LIN {X 0,Y 383.396,Z 1180.828,A -85,B 0,C 180,E1 16065.026,E2 16065.026} C_VEL
LIN {X 0,Y 390.535,Z 1171.867,A -85,B 0,C 180,E1 16063.935,E2 16063.935} C_VEL
LIN {X 0,Y 376.385,Z 1188.469,A -85,B 0,C 180,E1 16061.413,E2 16061.413} C_VEL
LIN {X 0,Y 362.666,Z 1204.614,A -85,B 0,C 180,E1 16058.341,E2 16058.341} C_VEL
LIN {X 0,Y 350.721,Z 1218.775,A -85,B 0,C 180,E1 16054.963,E2 16054.963} C_VEL
LIN {X 0,Y 340.496,Z 1230.965,A -85,B 0,C 180,E1 16051.317,E2 16051.317} C_VEL
LIN {X 0,Y 331.986,Z 1241.186,A -85,B 0,C 180,E1 16047.44,E2 16047.44} C_VEL
LIN {X 0,Y 325.156,Z 1249.467,A -85,B 0,C 180,E1 16043.371,E2 16043.371} C_VEL
LIN {X 0,Y 320.144,Z 1255.613,A -85,B 0,C 180,E1 16039.333,E2 16039.333} C_VEL
LIN {X 0,Y 316.54,Z 1259.979,A -85,B 0,C 180,E1 16035.2,E2 16035.2} C_VEL
LIN {X 0,Y 314.272,Z 1262.44,A -85,B 0,C 180,E1 16031.191,E2 16031.191} C_VEL
LIN {X 0,Y 312.948,Z 1263.309,A -85,B 0,C 180,E1 16026.974,E2 16026.974} C_VEL
LIN {X 0,Y 312.379,Z 1262.543,A -85,B 0,C 180,E1 16023.119,E2 16023.119} C_VEL
LIN {X 0,Y 312.208,Z 1260.385,A -85,B 0,C 180,E1 16019.633,E2 16019.633} C_VEL
LIN {X 0,Y 312.174,Z 1256.694,A -85,B 0,C 180,E1 16015.959,E2 16015.959} C_VEL
LIN {X 0,Y 312.386,Z 1251.681,A -85,B 0,C 180,E1 16012.459,E2 16012.459} C_VEL
LIN {X 0,Y 312.913,Z 1245.037,A -85,B 0,C 180,E1 16008.946,E2 16008.946} C_VEL
LIN {X 0,Y 313.943,Z 1236.737,A -85,B 0,C 180,E1 16005.427,E2 16005.427} C_VEL
LIN {X 0,Y 315.598,Z 1226.498,A -85,B 0,C 180,E1 16001.897,E2 16001.897} C_VEL
LIN {X 0,Y 317.811,Z 1214.873,A -85,B 0,C 180,E1 15998.595,E2 15998.595} C_VEL
LIN {X 0,Y 320.732,Z 1201.077,A -85,B 0,C 180,E1 15995.307,E2 15995.307} C_VEL
LIN {X 0,Y 324.178,Z 1185.749,A -85,B 0,C 180,E1 15992.242,E2 15992.242} C_VEL
LIN {X 0,Y 327.919,Z 1169.466,A -85,B 0,C 180,E1 15989.49,E2 15989.49} C_VEL
LIN {X 0,Y 332.099,Z 1150.975,A -85,B 0,C 180,E1 15986.862,E2 15986.862} C_VEL
LIN {X 0,Y 336.467,Z 1130.85,A -85,B 0,C 180,E1 15984.481,E2 15984.481} C_VEL
LIN {X 0,Y 340.596,Z 1110.333,A -85,B 0,C 180,E1 15982.46,E2 15982.46} C_VEL
LIN {X 0,Y 344.502,Z 1089.321,A -85,B 0,C 180,E1 15980.748,E2 15980.748} C_VEL
LIN {X 0,Y 348.276,Z 1066.302,A -85,B 0,C 180,E1 15979.221,E2 15979.221} C_VEL
LIN {X 0,Y 351.6,Z 1042.308,A -85,B 0,C 180,E1 15977.965,E2 15977.965} C_VEL
LIN {X 0,Y 354.32,Z 1018.528,A -85,B 0,C 180,E1 15977.027,E2 15977.027} C_VEL
LIN {X 0,Y 373.54,Z 802.907,A -85,B 0,C 180,E1 15971.161,E2 15971.161} C_VEL
LIN {X 0,Y 358.853,Z 773.867,A -85,B 0,C 180,E1 15968.29,E2 15968.29} C_VEL
LIN {X 0,Y 344.851,Z 748.162,A -85,B 0,C 180,E1 15965.343,E2 15965.343} C_VEL
LIN {X 0,Y 331.038,Z 724.458,A -85,B 0,C 180,E1 15962.193,E2 15962.193} C_VEL
LIN {X 0,Y 324.587,Z 713.661,A -85,B 0,C 180,E1 15960.552,E2 15960.552} C_VEL
LIN {X 0,Y 318.502,Z 700.77,A -85,B 0,C 180,E1 15957.485,E2 15957.485} C_VEL
LIN {X 0,Y 316.879,Z 697.207,A -85,B 0,C 180,E1 15956.622,E2 15956.622} C_VEL
LIN {X 0,Y 315.399,Z 693.796,A -85,B 0,C 180,E1 15955.795,E2 15955.795} C_VEL
LIN {X 0,Y 315.338,Z 693.386,A -85,B 0,C 180,E1 15955.658,E2 15955.658} C_VEL
LIN {X 0,Y 315.335,Z 693.387,A -85,B 0,C 180,E1 15951.193,E2 15951.193} C_VEL
LIN {X 0,Y 315.334,Z 693.384,A -85,B 0,C 180,E1 15946.741,E2 15946.741} C_VEL
LIN {X 0,Y 315.333,Z 693.371,A -85,B 0,C 180,E1 15942.268,E2 15942.268} C_VEL
LIN {X 0,Y 315.347,Z 693.369,A -85,B 0,C 180,E1 15937.655,E2 15937.655} C_VEL
LIN {X 0,Y 315.328,Z 693.376,A -85,B 0,C 180,E1 15933.093,E2 15933.093} C_VEL
LIN {X 0,Y 315.342,Z 693.38,A -85,B 0,C 180,E1 15928.549,E2 15928.549} C_VEL
LIN {X 0,Y 315.335,Z 693.391,A -85,B 0,C 180,E1 15923.996,E2 15923.996} C_VEL
LIN {X 0,Y 315.355,Z 693.532,A -85,B 0,C 180,E1 15921.478,E2 15921.478} C_VEL
LIN {X 0,Y 316.785,Z 697.081,A -85,B 0,C 180,E1 15920.189,E2 15920.189} C_VEL
LIN {X 0,Y 317.879,Z 698.667,A -85,B 0,C 180,E1 15919.491,E2 15919.491} C_VEL
LIN {X 0,Y 319.772,Z 702.458,A -85,B 0,C 180,E1 15918.093,E2 15918.093} C_VEL
LIN {X 0,Y 322.889,Z 708.89,A -85,B 0,C 180,E1 15915.842,E2 15915.842} C_VEL
LIN {X 0,Y 326.754,Z 716.586,A -85,B 0,C 180,E1 15913.286,E2 15913.286} C_VEL
LIN {X 0,Y 332.475,Z 729.013,A -85,B 0,C 180,E1 15909.585,E2 15909.585} C_VEL
LIN {X 0,Y 338.515,Z 742.871,A -85,B 0,C 180,E1 15905.883,E2 15905.883} C_VEL
LIN {X 0,Y 344.733,Z 758.436,A -85,B 0,C 180,E1 15902.165,E2 15902.165} C_VEL
LIN {X 0,Y 350.818,Z 775.213,A -85,B 0,C 180,E1 15898.565,E2 15898.565} C_VEL
LIN {X 0,Y 356.354,Z 792.064,A -85,B 0,C 180,E1 15895.281,E2 15895.281} C_VEL
LIN {X 0,Y 359.912,Z 803.987,A -85,B 0,C 180,E1 15893.128,E2 15893.128} C_VEL
LIN {X 0,Y 351.381,Z 845.901,A -85,B 0,C 180,E1 15888.452,E2 15888.452} C_VEL
LIN {X 0,Y 343.465,Z 888.943,A -85,B 0,C 180,E1 15883.627,E2 15883.627} C_VEL
LIN {X 0,Y 337.69,Z 924.781,A -85,B 0,C 180,E1 15879.624,E2 15879.624} C_VEL
LIN {X 0,Y 337.885,Z 936.89,A -85,B 0,C 180,E1 15879.108,E2 15879.108} C_VEL
LIN {X 0,Y 331.98,Z 1005.613,A -85,B 0,C 180,E1 15876.549,E2 15876.549} C_VEL
LIN {X 0,Y 327.912,Z 1055.103,A -85,B 0,C 180,E1 15874.422,E2 15874.422} C_VEL
LIN {X 0,Y 326.444,Z 1062.55,A -85,B 0,C 180,E1 15874.127,E2 15874.127} C_VEL
LIN {X 0,Y 319.464,Z 1081.052,A -85,B 0,C 180,E1 15873.458,E2 15873.458} C_VEL
LIN {X 0,Y 317.934,Z 1088.291,A -85,B 0,C 180,E1 15873.04,E2 15873.04} C_VEL
LIN {X 0,Y 316.347,Z 1105.042,A -85,B 0,C 180,E1 15871.724,E2 15871.724} C_VEL
LIN {X 0,Y 314.378,Z 1122.361,A -85,B 0,C 180,E1 15869.957,E2 15869.957} C_VEL
LIN {X 0,Y 312.544,Z 1137.053,A -85,B 0,C 180,E1 15868.053,E2 15868.053} C_VEL
LIN {X 0,Y 310.721,Z 1150.884,A -85,B 0,C 180,E1 15865.851,E2 15865.851} C_VEL
LIN {X 0,Y 308.968,Z 1164.225,A -85,B 0,C 180,E1 15863.216,E2 15863.216} C_VEL
LIN {X 0,Y 307.659,Z 1175.128,A -85,B 0,C 180,E1 15860.549,E2 15860.549} C_VEL
LIN {X 0,Y 306.728,Z 1184.712,A -85,B 0,C 180,E1 15857.648,E2 15857.648} C_VEL
LIN {X 0,Y 306.245,Z 1192.634,A -85,B 0,C 180,E1 15854.561,E2 15854.561} C_VEL
LIN {X 0,Y 306.245,Z 1198.64,A -85,B 0,C 180,E1 15851.488,E2 15851.488} C_VEL
LIN {X 0,Y 306.8,Z 1203.307,A -85,B 0,C 180,E1 15848.056,E2 15848.056} C_VEL
LIN {X 0,Y 307.938,Z 1205.89,A -85,B 0,C 180,E1 15844.843,E2 15844.843} C_VEL
LIN {X 0,Y 309.911,Z 1206.803,A -85,B 0,C 180,E1 15841.479,E2 15841.479} C_VEL
LIN {X 0,Y 312.741,Z 1205.82,A -85,B 0,C 180,E1 15838.168,E2 15838.168} C_VEL
LIN {X 0,Y 316.511,Z 1203.074,A -85,B 0,C 180,E1 15834.925,E2 15834.925} C_VEL
LIN {X 0,Y 321.273,Z 1198.385,A -85,B 0,C 180,E1 15831.748,E2 15831.748} C_VEL
LIN {X 0,Y 326.916,Z 1191.791,A -85,B 0,C 180,E1 15828.712,E2 15828.712} C_VEL
LIN {X 0,Y 333.133,Z 1183.559,A -85,B 0,C 180,E1 15825.929,E2 15825.929} C_VEL
LIN {X 0,Y 339.755,Z 1173.834,A -85,B 0,C 180,E1 15823.413,E2 15823.413} C_VEL
LIN {X 0,Y 346.624,Z 1162.742,A -85,B 0,C 180,E1 15821.151,E2 15821.151} C_VEL
LIN {X 0,Y 354.438,Z 1148.758,A -85,B 0,C 180,E1 15818.919,E2 15818.919} C_VEL
LIN {X 0,Y 362.13,Z 1133.307,A -85,B 0,C 180,E1 15817.002,E2 15817.002} C_VEL
LIN {X 0,Y 369.528,Z 1116.515,A -85,B 0,C 180,E1 15815.373,E2 15815.373} C_VEL
LIN {X 0,Y 377.955,Z 1095.177,A -85,B 0,C 180,E1 15813.781,E2 15813.781} C_VEL
LIN {X 0,Y 388.964,Z 1066.739,A -85,B 0,C 180,E1 15812.104,E2 15812.104} C_VEL
LIN {X 0,Y 400.416,Z 1034.438,A -85,B 0,C 180,E1 15810.606,E2 15810.606} C_VEL
LIN {X 0,Y 409.569,Z 1004.081,A -85,B 0,C 180,E1 15809.432,E2 15809.432} C_VEL
LIN {X 0,Y 415.633,Z 980.264,A -85,B 0,C 180,E1 15808.611,E2 15808.611} C_VEL
LIN {X 0,Y 419.158,Z 964.037,A -85,B 0,C 180,E1 15806.929,E2 15806.929} C_VEL
LIN {X 0,Y 419.266,Z 963.896,A -85,B 0,C 180,E1 15806.898,E2 15806.898} C_VEL
LIN {X 0,Y 415.267,Z 979.536,A -85,B 0,C 180,E1 15804.529,E2 15804.529} C_VEL
LIN {X 0,Y 413.402,Z 994.732,A -85,B 0,C 180,E1 15802.224,E2 15802.224} C_VEL
LIN {X 0,Y 406.081,Z 1023.051,A -85,B 0,C 180,E1 15801.76,E2 15801.76} C_VEL
LIN {X 0,Y 399.766,Z 1044.099,A -85,B 0,C 180,E1 15801.176,E2 15801.176} C_VEL
LIN {X 0,Y 391.3,Z 1069.63,A -85,B 0,C 180,E1 15800.125,E2 15800.125} C_VEL
LIN {X 0,Y 381.988,Z 1094.491,A -85,B 0,C 180,E1 15798.808,E2 15798.808} C_VEL
LIN {X 0,Y 372.816,Z 1116.783,A -85,B 0,C 180,E1 15797.292,E2 15797.292} C_VEL
LIN {X 0,Y 363.189,Z 1138.795,A -85,B 0,C 180,E1 15795.409,E2 15795.409} C_VEL
LIN {X 0,Y 353.773,Z 1158.891,A -85,B 0,C 180,E1 15793.263,E2 15793.263} C_VEL
LIN {X 0,Y 343.983,Z 1178.544,A -85,B 0,C 180,E1 15790.623,E2 15790.623} C_VEL
LIN {X 0,Y 335.047,Z 1195.941,A -85,B 0,C 180,E1 15787.715,E2 15787.715} C_VEL
LIN {X 0,Y 326.476,Z 1212.47,A -85,B 0,C 180,E1 15784.297,E2 15784.297} C_VEL
LIN {X 0,Y 319.092,Z 1227.195,A -85,B 0,C 180,E1 15780.503,E2 15780.503} C_VEL
LIN {X 0,Y 313.291,Z 1239.578,A -85,B 0,C 180,E1 15776.537,E2 15776.537} C_VEL
LIN {X 0,Y 308.935,Z 1250.237,A -85,B 0,C 180,E1 15772.231,E2 15772.231} C_VEL
LIN {X 0,Y 306.218,Z 1258.922,A -85,B 0,C 180,E1 15767.675,E2 15767.675} C_VEL
LIN {X 0,Y 305.799,Z 1260.852,A -85,B 0,C 180,E1 15766.524,E2 15766.524} C_VEL
LIN {X 0,Y 304.869,Z 1269.99,A -85,B 0,C 180,E1 15762.884,E2 15762.884} C_VEL
LIN {X 0,Y 304.511,Z 1277.274,A -85,B 0,C 180,E1 15759.256,E2 15759.256} C_VEL
LIN {X 0,Y 304.516,Z 1282.247,A -85,B 0,C 180,E1 15756.029,E2 15756.029} C_VEL
LIN {X 0,Y 304.597,Z 1286.195,A -85,B 0,C 180,E1 15752.443,E2 15752.443} C_VEL
LIN {X 0,Y 304.546,Z 1288.248,A -85,B 0,C 180,E1 15749.433,E2 15749.433} C_VEL
LIN {X 0,Y 304.303,Z 1289.341,A -85,B 0,C 180,E1 15745.852,E2 15745.852} C_VEL
LIN {X 0,Y 304.168,Z 1288.885,A -85,B 0,C 180,E1 15742.252,E2 15742.252} C_VEL
LIN {X 0,Y 304.527,Z 1286.905,A -85,B 0,C 180,E1 15738.252,E2 15738.252} C_VEL
LIN {X 0,Y 305.91,Z 1283.091,A -85,B 0,C 180,E1 15734.062,E2 15734.062} C_VEL
LIN {X 0,Y 308.723,Z 1277.309,A -85,B 0,C 180,E1 15729.721,E2 15729.721} C_VEL
LIN {X 0,Y 313.348,Z 1269.387,A -85,B 0,C 180,E1 15725.288,E2 15725.288} C_VEL
LIN {X 0,Y 319.828,Z 1259.544,A -85,B 0,C 180,E1 15721.013,E2 15721.013} C_VEL
LIN {X 0,Y 328.635,Z 1247.242,A -85,B 0,C 180,E1 15716.791,E2 15716.791} C_VEL
LIN {X 0,Y 339.52,Z 1232.892,A -85,B 0,C 180,E1 15712.861,E2 15712.861} C_VEL
LIN {X 0,Y 351.986,Z 1217.272,A -85,B 0,C 180,E1 15709.417,E2 15709.417} C_VEL
LIN {X 0,Y 366.387,Z 1199.946,A -85,B 0,C 180,E1 15706.332,E2 15706.332} C_VEL
LIN {X 0,Y 381.174,Z 1182.758,A -85,B 0,C 180,E1 15703.856,E2 15703.856} C_VEL
LIN {X 0,Y 366.383,Z 1198.617,A -85,B 0,C 180,E1 15701.126,E2 15701.126} C_VEL
LIN {X 0,Y 352.796,Z 1213.242,A -85,B 0,C 180,E1 15697.953,E2 15697.953} C_VEL
LIN {X 0,Y 340.964,Z 1226.045,A -85,B 0,C 180,E1 15694.471,E2 15694.471} C_VEL
LIN {X 0,Y 330.89,Z 1236.989,A -85,B 0,C 180,E1 15690.71,E2 15690.71} C_VEL
LIN {X 0,Y 322.245,Z 1246.426,A -85,B 0,C 180,E1 15686.54,E2 15686.54} C_VEL
LIN {X 0,Y 315.702,Z 1253.585,A -85,B 0,C 180,E1 15682.338,E2 15682.338} C_VEL
LIN {X 0,Y 310.997,Z 1258.719,A -85,B 0,C 180,E1 15678.172,E2 15678.172} C_VEL
LIN {X 0,Y 307.714,Z 1262.07,A -85,B 0,C 180,E1 15673.914,E2 15673.914} C_VEL
LIN {X 0,Y 305.744,Z 1263.639,A -85,B 0,C 180,E1 15669.791,E2 15669.791} C_VEL
LIN {X 0,Y 304.699,Z 1263.619,A -85,B 0,C 180,E1 15665.65,E2 15665.65} C_VEL
LIN {X 0,Y 304.294,Z 1262.122,A -85,B 0,C 180,E1 15661.883,E2 15661.883} C_VEL
LIN {X 0,Y 304.168,Z 1259.115,A -85,B 0,C 180,E1 15658.116,E2 15658.116} C_VEL
LIN {X 0,Y 304.229,Z 1254.904,A -85,B 0,C 180,E1 15654.531,E2 15654.531} C_VEL
LIN {X 0,Y 304.56,Z 1249.048,A -85,B 0,C 180,E1 15650.933,E2 15650.933} C_VEL
LIN {X 0,Y 305.361,Z 1241.165,A -85,B 0,C 180,E1 15647.134,E2 15647.134} C_VEL
LIN {X 0,Y 306.717,Z 1231.872,A -85,B 0,C 180,E1 15643.524,E2 15643.524} C_VEL
LIN {X 0,Y 308.79,Z 1220.431,A -85,B 0,C 180,E1 15639.897,E2 15639.897} C_VEL
LIN {X 0,Y 311.44,Z 1207.642,A -85,B 0,C 180,E1 15636.54,E2 15636.54} C_VEL
LIN {X 0,Y 314.645,Z 1193.344,A -85,B 0,C 180,E1 15633.38,E2 15633.38} C_VEL
LIN {X 0,Y 318.429,Z 1177.124,A -85,B 0,C 180,E1 15630.359,E2 15630.359} C_VEL
LIN {X 0,Y 322.444,Z 1159.96,A -85,B 0,C 180,E1 15627.661,E2 15627.661} C_VEL
LIN {X 0,Y 326.854,Z 1140.568,A -85,B 0,C 180,E1 15625.106,E2 15625.106} C_VEL
LIN {X 0,Y 331.363,Z 1119.567,A -85,B 0,C 180,E1 15622.811,E2 15622.811} C_VEL
LIN {X 0,Y 335.691,Z 1097.631,A -85,B 0,C 180,E1 15620.841,E2 15620.841} C_VEL
LIN {X 0,Y 339.457,Z 1076.238,A -85,B 0,C 180,E1 15619.273,E2 15619.273} C_VEL
LIN {X 0,Y 343.034,Z 1052.989,A -85,B 0,C 180,E1 15617.901,E2 15617.901} C_VEL
LIN {X 0,Y 346.115,Z 1028.65,A -85,B 0,C 180,E1 15616.79,E2 15616.79} C_VEL
LIN {X 0,Y 348.886,Z 1000.527,A -85,B 0,C 180,E1 15615.866,E2 15615.866} C_VEL
LIN {X 0,Y 366.833,Z 805.568,A -85,B 0,C 180,E1 15610.494,E2 15610.494} C_VEL
LIN {X 0,Y 352.729,Z 777.565,A -85,B 0,C 180,E1 15607.655,E2 15607.655} C_VEL
LIN {X 0,Y 339.122,Z 752.497,A -85,B 0,C 180,E1 15604.712,E2 15604.712} C_VEL
LIN {X 0,Y 325.773,Z 729.458,A -85,B 0,C 180,E1 15601.583,E2 15601.583} C_VEL
LIN {X 0,Y 316.726,Z 714.57,A -85,B 0,C 180,E1 15599.299,E2 15599.299} C_VEL
LIN {X 0,Y 310.669,Z 701.892,A -85,B 0,C 180,E1 15596.166,E2 15596.166} C_VEL
LIN {X 0,Y 309.075,Z 698.362,A -85,B 0,C 180,E1 15595.282,E2 15595.282} C_VEL
LIN {X 0,Y 307.473,Z 694.874,A -85,B 0,C 180,E1 15594.396,E2 15594.396} C_VEL
LIN {X 0,Y 307.397,Z 694.375,A -85,B 0,C 180,E1 15594.198,E2 15594.198} C_VEL
LIN {X 0,Y 307.401,Z 694.374,A -85,B 0,C 180,E1 15589.775,E2 15589.775} C_VEL
LIN {X 0,Y 307.395,Z 694.379,A -85,B 0,C 180,E1 15585.279,E2 15585.279} C_VEL
LIN {X 0,Y 307.399,Z 694.378,A -85,B 0,C 180,E1 15580.687,E2 15580.687} C_VEL
LIN {X 0,Y 307.404,Z 694.378,A -85,B 0,C 180,E1 15576.164,E2 15576.164} C_VEL
LIN {X 0,Y 307.393,Z 694.377,A -85,B 0,C 180,E1 15571.494,E2 15571.494} C_VEL
LIN {X 0,Y 307.39,Z 694.369,A -85,B 0,C 180,E1 15566.998,E2 15566.998} C_VEL
LIN {X 0,Y 307.402,Z 694.399,A -85,B 0,C 180,E1 15563.841,E2 15563.841} C_VEL
LIN {X 0,Y 308.662,Z 697.787,A -85,B 0,C 180,E1 15562.557,E2 15562.557} C_VEL
LIN {X 0,Y 309.997,Z 699.657,A -85,B 0,C 180,E1 15561.657,E2 15561.657} C_VEL
LIN {X 0,Y 311.768,Z 703.35,A -85,B 0,C 180,E1 15560.216,E2 15560.216} C_VEL
LIN {X 0,Y 312.888,Z 705.704,A -85,B 0,C 180,E1 15559.321,E2 15559.321} C_VEL
LIN {X 0,Y 315.072,Z 709.917,A -85,B 0,C 180,E1 15557.726,E2 15557.726} C_VEL
LIN {X 0,Y 317.516,Z 714.879,A -85,B 0,C 180,E1 15555.97,E2 15555.97} C_VEL
LIN {X 0,Y 321.344,Z 722.683,A -85,B 0,C 180,E1 15553.368,E2 15553.368} C_VEL
LIN {X 0,Y 326.788,Z 734.584,A -85,B 0,C 180,E1 15549.775,E2 15549.775} C_VEL
LIN {X 0,Y 332.659,Z 748.312,A -85,B 0,C 180,E1 15546.063,E2 15546.063} C_VEL
LIN {X 0,Y 338.777,Z 763.844,A -85,B 0,C 180,E1 15542.307,E2 15542.307} C_VEL
LIN {X 0,Y 344.667,Z 780.397,A -85,B 0,C 180,E1 15538.719,E2 15538.719} C_VEL
LIN {X 0,Y 350.147,Z 797.381,A -85,B 0,C 180,E1 15535.374,E2 15535.374} C_VEL
LIN {X 0,Y 352.858,Z 807.263,A -85,B 0,C 180,E1 15533.588,E2 15533.588} C_VEL
LIN {X 0,Y 344.019,Z 849.349,A -85,B 0,C 180,E1 15528.832,E2 15528.832} C_VEL
LIN {X 0,Y 336.014,Z 891.663,A -85,B 0,C 180,E1 15524.014,E2 15524.014} C_VEL
LIN {X 0,Y 330.403,Z 925.573,A -85,B 0,C 180,E1 15520.175,E2 15520.175} C_VEL
LIN {X 0,Y 330.552,Z 937.504,A -85,B 0,C 180,E1 15519.655,E2 15519.655} C_VEL
LIN {X 0,Y 324.763,Z 1002.82,A -85,B 0,C 180,E1 15517.166,E2 15517.166} C_VEL
LIN {X 0,Y 319.972,Z 1059.504,A -85,B 0,C 180,E1 15514.628,E2 15514.628} C_VEL
LIN {X 0,Y 318.293,Z 1083.967,A -85,B 0,C 180,E1 15513.326,E2 15513.326} C_VEL
LIN {X 0,Y 317.934,Z 1088.291,A -85,B 0,C 180,E1 15513.04,E2 15513.04} C_VEL
LIN {X 0,Y 316.33,Z 1095.446,A -85,B 0,C 180,E1 15512.568,E2 15512.568} C_VEL
LIN {X 0,Y 309.069,Z 1111.82,A -85,B 0,C 180,E1 15511.394,E2 15511.394} C_VEL
LIN {X 0,Y 307.076,Z 1118.46,A -85,B 0,C 180,E1 15510.737,E2 15510.737} C_VEL
LIN {X 0,Y 306.938,Z 1119.395,A -85,B 0,C 180,E1 15510.631,E2 15510.631} C_VEL
LIN {X 0,Y 304.937,Z 1135.362,A -85,B 0,C 180,E1 15508.603,E2 15508.603} C_VEL
LIN {X 0,Y 302.946,Z 1150.161,A -85,B 0,C 180,E1 15506.249,E2 15506.249} C_VEL
LIN {X 0,Y 301.316,Z 1162.312,A -85,B 0,C 180,E1 15503.882,E2 15503.882} C_VEL
LIN {X 0,Y 299.82,Z 1174.431,A -85,B 0,C 180,E1 15500.976,E2 15500.976} C_VEL
LIN {X 0,Y 298.846,Z 1183.869,A -85,B 0,C 180,E1 15498.129,E2 15498.129} C_VEL
LIN {X 0,Y 298.291,Z 1192.257,A -85,B 0,C 180,E1 15494.958,E2 15494.958} C_VEL
LIN {X 0,Y 298.252,Z 1198.949,A -85,B 0,C 180,E1 15491.604,E2 15491.604} C_VEL
LIN {X 0,Y 298.72,Z 1203.473,A -85,B 0,C 180,E1 15488.469,E2 15488.469} C_VEL
LIN {X 0,Y 299.991,Z 1206.779,A -85,B 0,C 180,E1 15484.779,E2 15484.779} C_VEL
LIN {X 0,Y 302.029,Z 1207.932,A -85,B 0,C 180,E1 15481.328,E2 15481.328} C_VEL
LIN {X 0,Y 304.977,Z 1207.303,A -85,B 0,C 180,E1 15477.933,E2 15477.933} C_VEL
LIN {X 0,Y 309.133,Z 1204.677,A -85,B 0,C 180,E1 15474.432,E2 15474.432} C_VEL
LIN {X 0,Y 314.705,Z 1199.678,A -85,B 0,C 180,E1 15470.859,E2 15470.859} C_VEL
LIN {X 0,Y 320.745,Z 1193.107,A -85,B 0,C 180,E1 15467.761,E2 15467.761} C_VEL
LIN {X 0,Y 326.925,Z 1185.524,A -85,B 0,C 180,E1 15465.113,E2 15465.113} C_VEL
LIN {X 0,Y 333.879,Z 1176.113,A -85,B 0,C 180,E1 15462.574,E2 15462.574} C_VEL
LIN {X 0,Y 342.055,Z 1163.724,A -85,B 0,C 180,E1 15460,E2 15460} C_VEL
LIN {X 0,Y 350.289,Z 1149.828,A -85,B 0,C 180,E1 15457.777,E2 15457.777} C_VEL
LIN {X 0,Y 358.08,Z 1135.171,A -85,B 0,C 180,E1 15455.94,E2 15455.94} C_VEL
LIN {X 0,Y 365.498,Z 1119.523,A -85,B 0,C 180,E1 15454.39,E2 15454.39} C_VEL
LIN {X 0,Y 373.522,Z 1100.646,A -85,B 0,C 180,E1 15452.93,E2 15452.93} C_VEL
LIN {X 0,Y 384.355,Z 1074.472,A -85,B 0,C 180,E1 15451.316,E2 15451.316} C_VEL
LIN {X 0,Y 394.683,Z 1047.623,A -85,B 0,C 180,E1 15450.005,E2 15450.005} C_VEL
LIN {X 0,Y 404.484,Z 1018.647,A -85,B 0,C 180,E1 15448.817,E2 15448.817} C_VEL
LIN {X 0,Y 412.96,Z 988.388,A -85,B 0,C 180,E1 15447.772,E2 15447.772} C_VEL
LIN {X 0,Y 414.238,Z 983.176,A -85,B 0,C 180,E1 15447.577,E2 15447.577} C_VEL
LIN {X 0,Y 415.981,Z 975.477,A -85,B 0,C 180,E1 15446.766,E2 15446.766} C_VEL
LIN {X 0,Y 411.85,Z 994.79,A -85,B 0,C 180,E1 15443.775,E2 15443.775} C_VEL
LIN {X 0,Y 411.359,Z 998.358,A -85,B 0,C 180,E1 15443.265,E2 15443.265} C_VEL
LIN {X 0,Y 404.458,Z 1023.469,A -85,B 0,C 180,E1 15442.866,E2 15442.866} C_VEL
LIN {X 0,Y 398.002,Z 1044.167,A -85,B 0,C 180,E1 15442.309,E2 15442.309} C_VEL
LIN {X 0,Y 389.393,Z 1068.851,A -85,B 0,C 180,E1 15441.313,E2 15441.313} C_VEL
LIN {X 0,Y 380.06,Z 1092.864,A -85,B 0,C 180,E1 15440.072,E2 15440.072} C_VEL
LIN {X 0,Y 370.536,Z 1115.069,A -85,B 0,C 180,E1 15438.602,E2 15438.602} C_VEL
LIN {X 0,Y 360.67,Z 1136.571,A -85,B 0,C 180,E1 15436.808,E2 15436.808} C_VEL
LIN {X 0,Y 351.165,Z 1155.855,A -85,B 0,C 180,E1 15434.803,E2 15434.803} C_VEL
LIN {X 0,Y 341.294,Z 1174.61,A -85,B 0,C 180,E1 15432.359,E2 15432.359} C_VEL
LIN {X 0,Y 331.635,Z 1192.202,A -85,B 0,C 180,E1 15429.503,E2 15429.503} C_VEL
LIN {X 0,Y 322.703,Z 1208.197,A -85,B 0,C 180,E1 15426.282,E2 15426.282} C_VEL
LIN {X 0,Y 315.1,Z 1222.005,A -85,B 0,C 180,E1 15422.859,E2 15422.859} C_VEL
LIN {X 0,Y 308.56,Z 1234.41,A -85,B 0,C 180,E1 15419.08,E2 15419.08} C_VEL
LIN {X 0,Y 303.16,Z 1245.717,A -85,B 0,C 180,E1 15414.76,E2 15414.76} C_VEL
LIN {X 0,Y 299.485,Z 1254.912,A -85,B 0,C 180,E1 15410.252,E2 15410.252} C_VEL
LIN {X 0,Y 297.668,Z 1261.534,A -85,B 0,C 180,E1 15406.116,E2 15406.116} C_VEL
LIN {X 0,Y 296.824,Z 1270.319,A -85,B 0,C 180,E1 15402.447,E2 15402.447} C_VEL
LIN {X 0,Y 296.533,Z 1277.393,A -85,B 0,C 180,E1 15398.725,E2 15398.725} C_VEL
LIN {X 0,Y 296.574,Z 1282.504,A -85,B 0,C 180,E1 15395.22,E2 15395.22} C_VEL
LIN {X 0,Y 296.635,Z 1285.986,A -85,B 0,C 180,E1 15391.736,E2 15391.736} C_VEL
LIN {X 0,Y 296.533,Z 1287.917,A -85,B 0,C 180,E1 15388.645,E2 15388.645} C_VEL
LIN {X 0,Y 296.261,Z 1288.828,A -85,B 0,C 180,E1 15384.963,E2 15384.963} C_VEL
LIN {X 0,Y 296.198,Z 1288.277,A -85,B 0,C 180,E1 15381.26,E2 15381.26} C_VEL
LIN {X 0,Y 296.889,Z 1285.861,A -85,B 0,C 180,E1 15376.736,E2 15376.736} C_VEL
LIN {X 0,Y 298.844,Z 1281.688,A -85,B 0,C 180,E1 15372.271,E2 15372.271} C_VEL
LIN {X 0,Y 302.415,Z 1275.546,A -85,B 0,C 180,E1 15367.787,E2 15367.787} C_VEL
LIN {X 0,Y 307.82,Z 1267.501,A -85,B 0,C 180,E1 15363.365,E2 15363.365} C_VEL
LIN {X 0,Y 315.588,Z 1257.086,A -85,B 0,C 180,E1 15358.904,E2 15358.904} C_VEL
LIN {X 0,Y 325.069,Z 1245.277,A -85,B 0,C 180,E1 15354.884,E2 15354.884} C_VEL
LIN {X 0,Y 337.249,Z 1230.907,A -85,B 0,C 180,E1 15350.968,E2 15350.968} C_VEL
LIN {X 0,Y 351.935,Z 1214.304,A -85,B 0,C 180,E1 15347.379,E2 15347.379} C_VEL
LIN {X 0,Y 367.323,Z 1197.534,A -85,B 0,C 180,E1 15344.503,E2 15344.503} C_VEL
LIN {X 0,Y 371.746,Z 1192.835,A -85,B 0,C 180,E1 15343.783,E2 15343.783} C_VEL
LIN {X 0,Y 356.342,Z 1207.941,A -85,B 0,C 180,E1 15340.829,E2 15340.829} C_VEL
LIN {X 0,Y 342.345,Z 1221.703,A -85,B 0,C 180,E1 15337.41,E2 15337.41} C_VEL
LIN {X 0,Y 330.725,Z 1233.151,A -85,B 0,C 180,E1 15333.8,E2 15333.8} C_VEL
LIN {X 0,Y 320.878,Z 1242.851,A -85,B 0,C 180,E1 15329.906,E2 15329.906} C_VEL
LIN {X 0,Y 312.514,Z 1251.09,A -85,B 0,C 180,E1 15325.59,E2 15325.59} C_VEL
LIN {X 0,Y 306.281,Z 1257.167,A -85,B 0,C 180,E1 15321.246,E2 15321.246} C_VEL
LIN {X 0,Y 301.901,Z 1261.314,A -85,B 0,C 180,E1 15316.945,E2 15316.945} C_VEL
LIN {X 0,Y 298.944,Z 1263.683,A -85,B 0,C 180,E1 15312.557,E2 15312.557} C_VEL
LIN {X 0,Y 297.289,Z 1264.352,A -85,B 0,C 180,E1 15308.316,E2 15308.316} C_VEL
LIN {X 0,Y 296.505,Z 1263.525,A -85,B 0,C 180,E1 15304.255,E2 15304.255} C_VEL
LIN {X 0,Y 296.223,Z 1261.196,A -85,B 0,C 180,E1 15300.387,E2 15300.387} C_VEL
LIN {X 0,Y 296.164,Z 1257.409,A -85,B 0,C 180,E1 15296.516,E2 15296.516} C_VEL
LIN {X 0,Y 296.345,Z 1252.342,A -85,B 0,C 180,E1 15292.828,E2 15292.828} C_VEL
LIN {X 0,Y 296.865,Z 1245.614,A -85,B 0,C 180,E1 15289.128,E2 15289.128} C_VEL
LIN {X 0,Y 297.98,Z 1236.72,A -85,B 0,C 180,E1 15285.225,E2 15285.225} C_VEL
LIN {X 0,Y 299.723,Z 1226.339,A -85,B 0,C 180,E1 15281.523,E2 15281.523} C_VEL
LIN {X 0,Y 302.238,Z 1213.777,A -85,B 0,C 180,E1 15277.843,E2 15277.843} C_VEL
LIN {X 0,Y 305.193,Z 1200.417,A -85,B 0,C 180,E1 15274.584,E2 15274.584} C_VEL
LIN {X 0,Y 308.861,Z 1184.803,A -85,B 0,C 180,E1 15271.371,E2 15271.371} C_VEL
LIN {X 0,Y 312.983,Z 1167.606,A -85,B 0,C 180,E1 15268.403,E2 15268.403} C_VEL
LIN {X 0,Y 317.11,Z 1150.123,A -85,B 0,C 180,E1 15265.857,E2 15265.857} C_VEL
LIN {X 0,Y 321.575,Z 1130.483,A -85,B 0,C 180,E1 15263.456,E2 15263.456} C_VEL
LIN {X 0,Y 326.096,Z 1108.982,A -85,B 0,C 180,E1 15261.28,E2 15261.28} C_VEL
LIN {X 0,Y 330.398,Z 1086.633,A -85,B 0,C 180,E1 15259.432,E2 15259.432} C_VEL
LIN {X 0,Y 334.204,Z 1063.994,A -85,B 0,C 180,E1 15257.919,E2 15257.919} C_VEL
LIN {X 0,Y 337.565,Z 1040.502,A -85,B 0,C 180,E1 15256.678,E2 15256.678} C_VEL
LIN {X 0,Y 340.425,Z 1016.058,A -85,B 0,C 180,E1 15255.708,E2 15255.708} C_VEL
LIN {X 0,Y 360.186,Z 808.245,A -85,B 0,C 180,E1 15249.811,E2 15249.811} C_VEL
LIN {X 0,Y 345.847,Z 779.769,A -85,B 0,C 180,E1 15246.84,E2 15246.84} C_VEL
LIN {X 0,Y 332.04,Z 754.342,A -85,B 0,C 180,E1 15243.754,E2 15243.754} C_VEL
LIN {X 0,Y 318.289,Z 730.723,A -85,B 0,C 180,E1 15240.411,E2 15240.411} C_VEL
LIN {X 0,Y 308.508,Z 714.884,A -85,B 0,C 180,E1 15237.823,E2 15237.823} C_VEL
LIN {X 0,Y 303.238,Z 703.637,A -85,B 0,C 180,E1 15234.967,E2 15234.967} C_VEL
LIN {X 0,Y 300.892,Z 699.021,A -85,B 0,C 180,E1 15233.711,E2 15233.711} C_VEL
LIN {X 0,Y 299.472,Z 695.441,A -85,B 0,C 180,E1 15232.813,E2 15232.813} C_VEL
LIN {X 0,Y 299.465,Z 695.366,A -85,B 0,C 180,E1 15228.294,E2 15228.294} C_VEL
LIN {X 0,Y 299.456,Z 695.346,A -85,B 0,C 180,E1 15223.673,E2 15223.673} C_VEL
LIN {X 0,Y 299.451,Z 695.35,A -85,B 0,C 180,E1 15219.225,E2 15219.225} C_VEL
LIN {X 0,Y 299.451,Z 695.352,A -85,B 0,C 180,E1 15214.791,E2 15214.791} C_VEL
LIN {X 0,Y 299.474,Z 695.347,A -85,B 0,C 180,E1 15210.194,E2 15210.194} C_VEL
LIN {X 0,Y 299.474,Z 695.525,A -85,B 0,C 180,E1 15206.366,E2 15206.366} C_VEL
LIN {X 0,Y 300.928,Z 699.075,A -85,B 0,C 180,E1 15204.856,E2 15204.856} C_VEL
LIN {X 0,Y 302.19,Z 700.87,A -85,B 0,C 180,E1 15203.925,E2 15203.925} C_VEL
LIN {X 0,Y 304.183,Z 704.746,A -85,B 0,C 180,E1 15202.257,E2 15202.257} C_VEL
LIN {X 0,Y 307.339,Z 711.107,A -85,B 0,C 180,E1 15199.695,E2 15199.695} C_VEL
LIN {X 0,Y 309.935,Z 716.357,A -85,B 0,C 180,E1 15197.709,E2 15197.709} C_VEL
LIN {X 0,Y 313.471,Z 723.305,A -85,B 0,C 180,E1 15195.219,E2 15195.219} C_VEL
LIN {X 0,Y 319.019,Z 735.392,A -85,B 0,C 180,E1 15191.358,E2 15191.358} C_VEL
LIN {X 0,Y 325.045,Z 749.369,A -85,B 0,C 180,E1 15187.389,E2 15187.389} C_VEL
LIN {X 0,Y 330.934,Z 764.239,A -85,B 0,C 180,E1 15183.634,E2 15183.634} C_VEL
LIN {X 0,Y 336.892,Z 780.729,A -85,B 0,C 180,E1 15179.898,E2 15179.898} C_VEL
LIN {X 0,Y 342.575,Z 798.244,A -85,B 0,C 180,E1 15176.323,E2 15176.323} C_VEL
LIN {X 0,Y 345.878,Z 810.106,A -85,B 0,C 180,E1 15174.116,E2 15174.116} C_VEL
LIN {X 0,Y 337.014,Z 851.085,A -85,B 0,C 180,E1 15169.423,E2 15169.423} C_VEL
LIN {X 0,Y 328.686,Z 893.769,A -85,B 0,C 180,E1 15164.489,E2 15164.489} C_VEL
LIN {X 0,Y 323.125,Z 926.24,A -85,B 0,C 180,E1 15160.748,E2 15160.748} C_VEL
LIN {X 0,Y 323.236,Z 938.083,A -85,B 0,C 180,E1 15160.222,E2 15160.222} C_VEL
LIN {X 0,Y 317.116,Z 1004.653,A -85,B 0,C 180,E1 15157.596,E2 15157.596} C_VEL
LIN {X 0,Y 312.335,Z 1059.503,A -85,B 0,C 180,E1 15155.061,E2 15155.061} C_VEL
LIN {X 0,Y 310.574,Z 1084.314,A -85,B 0,C 180,E1 15153.706,E2 15153.706} C_VEL
LIN {X 0,Y 309.07,Z 1100.675,A -85,B 0,C 180,E1 15152.482,E2 15152.482} C_VEL
LIN {X 0,Y 307.168,Z 1117.511,A -85,B 0,C 180,E1 15150.844,E2 15150.844} C_VEL
LIN {X 0,Y 306.938,Z 1119.395,A -85,B 0,C 180,E1 15150.631,E2 15150.631} C_VEL
LIN {X 0,Y 305.165,Z 1125.905,A -85,B 0,C 180,E1 15149.898,E2 15149.898} C_VEL
LIN {X 0,Y 297.26,Z 1141.398,A -85,B 0,C 180,E1 15147.973,E2 15147.973} C_VEL
LIN {X 0,Y 295.486,Z 1147.262,A -85,B 0,C 180,E1 15147.05,E2 15147.05} C_VEL
LIN {X 0,Y 293.614,Z 1160.892,A -85,B 0,C 180,E1 15144.442,E2 15144.442} C_VEL
LIN {X 0,Y 292.107,Z 1172.494,A -85,B 0,C 180,E1 15141.696,E2 15141.696} C_VEL
LIN {X 0,Y 290.982,Z 1182.946,A -85,B 0,C 180,E1 15138.637,E2 15138.637} C_VEL
LIN {X 0,Y 290.364,Z 1191.248,A -85,B 0,C 180,E1 15135.581,E2 15135.581} C_VEL
LIN {X 0,Y 290.226,Z 1198.167,A -85,B 0,C 180,E1 15132.334,E2 15132.334} C_VEL
LIN {X 0,Y 290.638,Z 1203.46,A -85,B 0,C 180,E1 15128.906,E2 15128.906} C_VEL
LIN {X 0,Y 291.689,Z 1207.022,A -85,B 0,C 180,E1 15125.508,E2 15125.508} C_VEL
LIN {X 0,Y 293.598,Z 1208.883,A -85,B 0,C 180,E1 15121.952,E2 15121.952} C_VEL
LIN {X 0,Y 296.444,Z 1208.955,A -85,B 0,C 180,E1 15118.454,E2 15118.454} C_VEL
LIN {X 0,Y 300.516,Z 1207.09,A -85,B 0,C 180,E1 15114.846,E2 15114.846} C_VEL
LIN {X 0,Y 305.73,Z 1203.199,A -85,B 0,C 180,E1 15111.347,E2 15111.347} C_VEL
LIN {X 0,Y 311.717,Z 1197.607,A -85,B 0,C 180,E1 15108.153,E2 15108.153} C_VEL
LIN {X 0,Y 318.284,Z 1190.521,A -85,B 0,C 180,E1 15105.258,E2 15105.258} C_VEL
LIN {X 0,Y 325.725,Z 1181.46,A -85,B 0,C 180,E1 15102.492,E2 15102.492} C_VEL
LIN {X 0,Y 334.021,Z 1170.197,A -85,B 0,C 180,E1 15099.864,E2 15099.864} C_VEL
LIN {X 0,Y 342.634,Z 1157.188,A -85,B 0,C 180,E1 15097.524,E2 15097.524} C_VEL
LIN {X 0,Y 351.442,Z 1142.322,A -85,B 0,C 180,E1 15095.456,E2 15095.456} C_VEL
LIN {X 0,Y 359.991,Z 1126.098,A -85,B 0,C 180,E1 15093.703,E2 15093.703} C_VEL
LIN {X 0,Y 368.164,Z 1108.593,A -85,B 0,C 180,E1 15092.24,E2 15092.24} C_VEL
LIN {X 0,Y 379.88,Z 1082.116,A -85,B 0,C 180,E1 15090.514,E2 15090.514} C_VEL
LIN {X 0,Y 391.402,Z 1054.205,A -85,B 0,C 180,E1 15089.104,E2 15089.104} C_VEL
LIN {X 0,Y 402.626,Z 1022.862,A -85,B 0,C 180,E1 15087.812,E2 15087.812} C_VEL
LIN {X 0,Y 411.006,Z 994.494,A -85,B 0,C 180,E1 15086.831,E2 15086.831} C_VEL
LIN {X 0,Y 412.898,Z 987.241,A -85,B 0,C 180,E1 15086.59,E2 15086.59} C_VEL
LIN {X 0,Y 409.602,Z 1001.891,A -85,B 0,C 180,E1 15084.33,E2 15084.33} C_VEL
LIN {X 0,Y 401.881,Z 1028.275,A -85,B 0,C 180,E1 15083.895,E2 15083.895} C_VEL
LIN {X 0,Y 395.205,Z 1048.298,A -85,B 0,C 180,E1 15083.32,E2 15083.32} C_VEL
LIN {X 0,Y 385.272,Z 1074.944,A -85,B 0,C 180,E1 15082.206,E2 15082.206} C_VEL
LIN {X 0,Y 375.375,Z 1098.477,A -85,B 0,C 180,E1 15080.934,E2 15080.934} C_VEL
LIN {X 0,Y 365.699,Z 1119.751,A -85,B 0,C 180,E1 15079.469,E2 15079.469} C_VEL
LIN {X 0,Y 354.646,Z 1142.299,A -85,B 0,C 180,E1 15077.495,E2 15077.495} C_VEL
LIN {X 0,Y 344.024,Z 1162.093,A -85,B 0,C 180,E1 15075.282,E2 15075.282} C_VEL
LIN {X 0,Y 333.437,Z 1180.617,A -85,B 0,C 180,E1 15072.661,E2 15072.661} C_VEL
LIN {X 0,Y 323.186,Z 1197.89,A -85,B 0,C 180,E1 15069.589,E2 15069.589} C_VEL
LIN {X 0,Y 313.781,Z 1213.506,A -85,B 0,C 180,E1 15066.119,E2 15066.119} C_VEL
LIN {X 0,Y 305.227,Z 1228.034,A -85,B 0,C 180,E1 15062.049,E2 15062.049} C_VEL
LIN {X 0,Y 298.487,Z 1240.168,A -85,B 0,C 180,E1 15057.748,E2 15057.748} C_VEL
LIN {X 0,Y 293.45,Z 1250.458,A -85,B 0,C 180,E1 15053.066,E2 15053.066} C_VEL
LIN {X 0,Y 290.408,Z 1258.453,A -85,B 0,C 180,E1 15048.256,E2 15048.256} C_VEL
LIN {X 0,Y 289.595,Z 1261.756,A -85,B 0,C 180,E1 15045.826,E2 15045.826} C_VEL
LIN {X 0,Y 288.819,Z 1270.16,A -85,B 0,C 180,E1 15042.189,E2 15042.189} C_VEL
LIN {X 0,Y 288.57,Z 1277.16,A -85,B 0,C 180,E1 15038.365,E2 15038.365} C_VEL
LIN {X 0,Y 288.627,Z 1282.205,A -85,B 0,C 180,E1 15034.766,E2 15034.766} C_VEL
LIN {X 0,Y 288.676,Z 1285.599,A -85,B 0,C 180,E1 15031.188,E2 15031.188} C_VEL
LIN {X 0,Y 288.519,Z 1287.467,A -85,B 0,C 180,E1 15028.011,E2 15028.011} C_VEL
LIN {X 0,Y 288.23,Z 1288.302,A -85,B 0,C 180,E1 15024.024,E2 15024.024} C_VEL
LIN {X 0,Y 288.273,Z 1287.628,A -85,B 0,C 180,E1 15020.088,E2 15020.088} C_VEL
LIN {X 0,Y 289.245,Z 1285.168,A -85,B 0,C 180,E1 15015.585,E2 15015.585} C_VEL
LIN {X 0,Y 291.632,Z 1280.937,A -85,B 0,C 180,E1 15010.989,E2 15010.989} C_VEL
LIN {X 0,Y 295.898,Z 1274.634,A -85,B 0,C 180,E1 15006.287,E2 15006.287} C_VEL
LIN {X 0,Y 302.111,Z 1266.499,A -85,B 0,C 180,E1 15001.75,E2 15001.75} C_VEL
LIN {X 0,Y 311.107,Z 1255.734,A -85,B 0,C 180,E1 14997.098,E2 14997.098} C_VEL
LIN {X 0,Y 322.479,Z 1243.018,A -85,B 0,C 180,E1 14992.796,E2 14992.796} C_VEL
LIN {X 0,Y 335.613,Z 1229.085,A -85,B 0,C 180,E1 14989.044,E2 14989.044} C_VEL
LIN {X 0,Y 350.853,Z 1213.497,A -85,B 0,C 180,E1 14985.713,E2 14985.713} C_VEL
LIN {X 0,Y 362.185,Z 1202.23,A -85,B 0,C 180,E1 14983.699,E2 14983.699} C_VEL
LIN {X 0,Y 346.234,Z 1216.524,A -85,B 0,C 180,E1 14980.525,E2 14980.525} C_VEL
LIN {X 0,Y 332.377,Z 1228.929,A -85,B 0,C 180,E1 14976.989,E2 14976.989} C_VEL
LIN {X 0,Y 320.451,Z 1239.587,A -85,B 0,C 180,E1 14973.096,E2 14973.096} C_VEL
LIN {X 0,Y 310.495,Z 1248.431,A -85,B 0,C 180,E1 14968.885,E2 14968.885} C_VEL
LIN {X 0,Y 302.517,Z 1255.435,A -85,B 0,C 180,E1 14964.403,E2 14964.403} C_VEL
LIN {X 0,Y 296.484,Z 1260.542,A -85,B 0,C 180,E1 14959.709,E2 14959.709} C_VEL
LIN {X 0,Y 292.593,Z 1263.571,A -85,B 0,C 180,E1 14955.256,E2 14955.256} C_VEL
LIN {X 0,Y 290.108,Z 1264.869,A -85,B 0,C 180,E1 14950.726,E2 14950.726} C_VEL
LIN {X 0,Y 288.835,Z 1264.464,A -85,B 0,C 180,E1 14946.36,E2 14946.36} C_VEL
LIN {X 0,Y 288.312,Z 1262.588,A -85,B 0,C 180,E1 14942.186,E2 14942.186} C_VEL
LIN {X 0,Y 288.17,Z 1259.462,A -85,B 0,C 180,E1 14938.409,E2 14938.409} C_VEL
LIN {X 0,Y 288.234,Z 1254.663,A -85,B 0,C 180,E1 14934.426,E2 14934.426} C_VEL
LIN {X 0,Y 288.6,Z 1248.585,A -85,B 0,C 180,E1 14930.628,E2 14930.628} C_VEL
LIN {X 0,Y 289.428,Z 1240.719,A -85,B 0,C 180,E1 14926.82,E2 14926.82} C_VEL
LIN {X 0,Y 290.999,Z 1230.459,A -85,B 0,C 180,E1 14922.796,E2 14922.796} C_VEL
LIN {X 0,Y 293.262,Z 1218.72,A -85,B 0,C 180,E1 14919.022,E2 14919.022} C_VEL
LIN {X 0,Y 296.008,Z 1206.246,A -85,B 0,C 180,E1 14915.663,E2 14915.663} C_VEL
LIN {X 0,Y 299.469,Z 1191.493,A -85,B 0,C 180,E1 14912.348,E2 14912.348} C_VEL
LIN {X 0,Y 303.404,Z 1175.307,A -85,B 0,C 180,E1 14909.282,E2 14909.282} C_VEL
LIN {X 0,Y 307.857,Z 1157.025,A -85,B 0,C 180,E1 14906.374,E2 14906.374} C_VEL
LIN {X 0,Y 312.562,Z 1137.027,A -85,B 0,C 180,E1 14903.725,E2 14903.725} C_VEL
LIN {X 0,Y 317.097,Z 1116.635,A -85,B 0,C 180,E1 14901.479,E2 14901.479} C_VEL
LIN {X 0,Y 321.409,Z 1095.64,A -85,B 0,C 180,E1 14899.561,E2 14899.561} C_VEL
LIN {X 0,Y 325.608,Z 1072.718,A -85,B 0,C 180,E1 14897.857,E2 14897.857} C_VEL
LIN {X 0,Y 329.377,Z 1048.583,A -85,B 0,C 180,E1 14896.44,E2 14896.44} C_VEL
LIN {X 0,Y 332.597,Z 1023.342,A -85,B 0,C 180,E1 14895.316,E2 14895.316} C_VEL
LIN {X 0,Y 336.519,Z 982.47,A -85,B 0,C 180,E1 14894.032,E2 14894.032} C_VEL
LIN {X 0,Y 353.512,Z 810.867,A -85,B 0,C 180,E1 14889.107,E2 14889.107} C_VEL
LIN {X 0,Y 339.578,Z 783.176,A -85,B 0,C 180,E1 14886.133,E2 14886.133} C_VEL
LIN {X 0,Y 326.322,Z 758.638,A -85,B 0,C 180,E1 14883.081,E2 14883.081} C_VEL
LIN {X 0,Y 312.721,Z 735.138,A -85,B 0,C 180,E1 14879.685,E2 14879.685} C_VEL
LIN {X 0,Y 301.25,Z 716.693,A -85,B 0,C 180,E1 14876.57,E2 14876.57} C_VEL
LIN {X 0,Y 300.045,Z 714.469,A -85,B 0,C 180,E1 14876.099,E2 14876.099} C_VEL
LIN {X 0,Y 295.078,Z 704.252,A -85,B 0,C 180,E1 14873.36,E2 14873.36} C_VEL
LIN {X 0,Y 293.14,Z 700.273,A -85,B 0,C 180,E1 14872.25,E2 14872.25} C_VEL
LIN {X 0,Y 291.604,Z 696.883,A -85,B 0,C 180,E1 14871.316,E2 14871.316} C_VEL
LIN {X 0,Y 291.52,Z 696.354,A -85,B 0,C 180,E1 14871.102,E2 14871.102} C_VEL
LIN {X 0,Y 291.518,Z 696.35,A -85,B 0,C 180,E1 14866.543,E2 14866.543} C_VEL
LIN {X 0,Y 291.514,Z 696.34,A -85,B 0,C 180,E1 14861.879,E2 14861.879} C_VEL
LIN {X 0,Y 291.527,Z 696.339,A -85,B 0,C 180,E1 14857.293,E2 14857.293} C_VEL
LIN {X 0,Y 291.512,Z 696.347,A -85,B 0,C 180,E1 14852.558,E2 14852.558} C_VEL
LIN {X 0,Y 291.539,Z 696.503,A -85,B 0,C 180,E1 14849.217,E2 14849.217} C_VEL
LIN {X 0,Y 292.854,Z 699.888,A -85,B 0,C 180,E1 14847.655,E2 14847.655} C_VEL
LIN {X 0,Y 294.314,Z 701.888,A -85,B 0,C 180,E1 14846.497,E2 14846.497} C_VEL
LIN {X 0,Y 296.219,Z 705.686,A -85,B 0,C 180,E1 14844.736,E2 14844.736} C_VEL
LIN {X 0,Y 297.039,Z 707.236,A -85,B 0,C 180,E1 14844.013,E2 14844.013} C_VEL
LIN {X 0,Y 299.489,Z 711.983,A -85,B 0,C 180,E1 14841.942,E2 14841.942} C_VEL
LIN {X 0,Y 301.982,Z 716.996,A -85,B 0,C 180,E1 14839.896,E2 14839.896} C_VEL
LIN {X 0,Y 305.871,Z 724.655,A -85,B 0,C 180,E1 14836.967,E2 14836.967} C_VEL
LIN {X 0,Y 311.318,Z 736.312,A -85,B 0,C 180,E1 14833.009,E2 14833.009} C_VEL
LIN {X 0,Y 316.932,Z 749.314,A -85,B 0,C 180,E1 14829.117,E2 14829.117} C_VEL
LIN {X 0,Y 322.46,Z 762.991,A -85,B 0,C 180,E1 14825.452,E2 14825.452} C_VEL
LIN {X 0,Y 328.075,Z 778.092,A -85,B 0,C 180,E1 14821.813,E2 14821.813} C_VEL
LIN {X 0,Y 333.691,Z 794.87,A -85,B 0,C 180,E1 14818.175,E2 14818.175} C_VEL
LIN {X 0,Y 338.978,Z 812.526,A -85,B 0,C 180,E1 14814.709,E2 14814.709} C_VEL
LIN {X 0,Y 330.034,Z 852.703,A -85,B 0,C 180,E1 14810.041,E2 14810.041} C_VEL
LIN {X 0,Y 321.459,Z 895.291,A -85,B 0,C 180,E1 14805.043,E2 14805.043} C_VEL
LIN {X 0,Y 315.853,Z 926.96,A -85,B 0,C 180,E1 14801.333,E2 14801.333} C_VEL
LIN {X 0,Y 315.915,Z 938.584,A -85,B 0,C 180,E1 14800.8,E2 14800.8} C_VEL
LIN {X 0,Y 309.607,Z 1005.218,A -85,B 0,C 180,E1 14798.101,E2 14798.101} C_VEL
LIN {X 0,Y 304.707,Z 1059.606,A -85,B 0,C 180,E1 14795.509,E2 14795.509} C_VEL
LIN {X 0,Y 302.825,Z 1084.809,A -85,B 0,C 180,E1 14794.074,E2 14794.074} C_VEL
LIN {X 0,Y 301.204,Z 1101.775,A -85,B 0,C 180,E1 14792.759,E2 14792.759} C_VEL
LIN {X 0,Y 299.232,Z 1118.766,A -85,B 0,C 180,E1 14791.052,E2 14791.052} C_VEL
LIN {X 0,Y 297.168,Z 1134.912,A -85,B 0,C 180,E1 14788.981,E2 14788.981} C_VEL
LIN {X 0,Y 295.486,Z 1147.262,A -85,B 0,C 180,E1 14787.05,E2 14787.05} C_VEL
LIN {X 0,Y 293.732,Z 1152.927,A -85,B 0,C 180,E1 14786.073,E2 14786.073} C_VEL
LIN {X 0,Y 285.986,Z 1166.101,A -85,B 0,C 180,E1 14783.476,E2 14783.476} C_VEL
LIN {X 0,Y 284.363,Z 1170.973,A -85,B 0,C 180,E1 14782.303,E2 14782.303} C_VEL
LIN {X 0,Y 283.196,Z 1181.234,A -85,B 0,C 180,E1 14779.384,E2 14779.384} C_VEL
LIN {X 0,Y 282.429,Z 1190.647,A -85,B 0,C 180,E1 14776.03,E2 14776.03} C_VEL
LIN {X 0,Y 282.225,Z 1197.886,A -85,B 0,C 180,E1 14772.689,E2 14772.689} C_VEL
LIN {X 0,Y 282.601,Z 1203.647,A -85,B 0,C 180,E1 14769.162,E2 14769.162} C_VEL
LIN {X 0,Y 283.717,Z 1207.705,A -85,B 0,C 180,E1 14765.46,E2 14765.46} C_VEL
LIN {X 0,Y 285.693,Z 1209.901,A -85,B 0,C 180,E1 14761.805,E2 14761.805} C_VEL
LIN {X 0,Y 288.839,Z 1210.249,A -85,B 0,C 180,E1 14758.016,E2 14758.016} C_VEL
LIN {X 0,Y 293.12,Z 1208.602,A -85,B 0,C 180,E1 14754.323,E2 14754.323} C_VEL
LIN {X 0,Y 298.275,Z 1205.239,A -85,B 0,C 180,E1 14750.935,E2 14750.935} C_VEL
LIN {X 0,Y 304.482,Z 1200.073,A -85,B 0,C 180,E1 14747.675,E2 14747.675} C_VEL
LIN {X 0,Y 312.133,Z 1192.517,A -85,B 0,C 180,E1 14744.39,E2 14744.39} C_VEL
LIN {X 0,Y 320.414,Z 1183.165,A -85,B 0,C 180,E1 14741.44,E2 14741.44} C_VEL
LIN {X 0,Y 329.664,Z 1171.407,A -85,B 0,C 180,E1 14738.656,E2 14738.656} C_VEL
LIN {X 0,Y 338.729,Z 1158.527,A -85,B 0,C 180,E1 14736.331,E2 14736.331} C_VEL
LIN {X 0,Y 347.964,Z 1143.876,A -85,B 0,C 180,E1 14734.284,E2 14734.284} C_VEL
LIN {X 0,Y 356.908,Z 1127.977,A -85,B 0,C 180,E1 14732.558,E2 14732.558} C_VEL
LIN {X 0,Y 365.315,Z 1111.162,A -85,B 0,C 180,E1 14731.141,E2 14731.141} C_VEL
LIN {X 0,Y 377.195,Z 1085.983,A -85,B 0,C 180,E1 14729.483,E2 14729.483} C_VEL
LIN {X 0,Y 388.943,Z 1058.996,A -85,B 0,C 180,E1 14728.109,E2 14728.109} C_VEL
LIN {X 0,Y 399.636,Z 1030.992,A -85,B 0,C 180,E1 14726.945,E2 14726.945} C_VEL
LIN {X 0,Y 408.427,Z 1003.806,A -85,B 0,C 180,E1 14725.985,E2 14725.985} C_VEL
LIN {X 0,Y 408.913,Z 1002.147,A -85,B 0,C 180,E1 14725.904,E2 14725.904} C_VEL
LIN {X 0,Y 408.046,Z 1005.476,A -85,B 0,C 180,E1 14725.409,E2 14725.409} C_VEL
LIN {X 0,Y 400.615,Z 1029.709,A -85,B 0,C 180,E1 14725.008,E2 14725.008} C_VEL
LIN {X 0,Y 393.392,Z 1050.273,A -85,B 0,C 180,E1 14724.42,E2 14724.42} C_VEL
LIN {X 0,Y 383.636,Z 1075.264,A -85,B 0,C 180,E1 14723.389,E2 14723.389} C_VEL
LIN {X 0,Y 373.098,Z 1099.325,A -85,B 0,C 180,E1 14722.111,E2 14722.111} C_VEL
LIN {X 0,Y 362.757,Z 1120.874,A -85,B 0,C 180,E1 14720.634,E2 14720.634} C_VEL
LIN {X 0,Y 352.345,Z 1141.11,A -85,B 0,C 180,E1 14718.885,E2 14718.885} C_VEL
LIN {X 0,Y 341.23,Z 1160.752,A -85,B 0,C 180,E1 14716.729,E2 14716.729} C_VEL
LIN {X 0,Y 330.081,Z 1179.117,A -85,B 0,C 180,E1 14714.16,E2 14714.16} C_VEL
LIN {X 0,Y 319.186,Z 1196.255,A -85,B 0,C 180,E1 14711.132,E2 14711.132} C_VEL
LIN {X 0,Y 309.12,Z 1211.771,A -85,B 0,C 180,E1 14707.683,E2 14707.683} C_VEL
LIN {X 0,Y 299.816,Z 1226.236,A -85,B 0,C 180,E1 14703.611,E2 14703.611} C_VEL
LIN {X 0,Y 292.368,Z 1238.355,A -85,B 0,C 180,E1 14699.275,E2 14699.275} C_VEL
LIN {X 0,Y 286.851,Z 1248.283,A -85,B 0,C 180,E1 14694.723,E2 14694.723} C_VEL
LIN {X 0,Y 283.366,Z 1255.858,A -85,B 0,C 180,E1 14690.228,E2 14690.228} C_VEL
LIN {X 0,Y 281.506,Z 1262.107,A -85,B 0,C 180,E1 14685.447,E2 14685.447} C_VEL
LIN {X 0,Y 280.786,Z 1270.453,A -85,B 0,C 180,E1 14681.681,E2 14681.681} C_VEL
LIN {X 0,Y 280.615,Z 1277.06,A -85,B 0,C 180,E1 14677.871,E2 14677.871} C_VEL
LIN {X 0,Y 280.682,Z 1281.866,A -85,B 0,C 180,E1 14674.287,E2 14674.287} C_VEL
LIN {X 0,Y 280.707,Z 1285.185,A -85,B 0,C 180,E1 14670.61,E2 14670.61} C_VEL
LIN {X 0,Y 280.483,Z 1287.082,A -85,B 0,C 180,E1 14667.137,E2 14667.137} C_VEL
LIN {X 0,Y 280.208,Z 1287.76,A -85,B 0,C 180,E1 14663.029,E2 14663.029} C_VEL
LIN {X 0,Y 280.412,Z 1286.989,A -85,B 0,C 180,E1 14658.896,E2 14658.896} C_VEL
LIN {X 0,Y 281.792,Z 1284.323,A -85,B 0,C 180,E1 14654.141,E2 14654.141} C_VEL
LIN {X 0,Y 284.908,Z 1279.755,A -85,B 0,C 180,E1 14649.237,E2 14649.237} C_VEL
LIN {X 0,Y 289.954,Z 1273.409,A -85,B 0,C 180,E1 14644.463,E2 14644.463} C_VEL
LIN {X 0,Y 297.368,Z 1264.872,A -85,B 0,C 180,E1 14639.708,E2 14639.708} C_VEL
LIN {X 0,Y 307.036,Z 1254.56,A -85,B 0,C 180,E1 14635.254,E2 14635.254} C_VEL
LIN {X 0,Y 319.951,Z 1241.573,A -85,B 0,C 180,E1 14630.853,E2 14630.853} C_VEL
LIN {X 0,Y 334.787,Z 1227.368,A -85,B 0,C 180,E1 14627.079,E2 14627.079} C_VEL
LIN {X 0,Y 351.144,Z 1212.209,A -85,B 0,C 180,E1 14623.908,E2 14623.908} C_VEL
LIN {X 0,Y 352.631,Z 1210.863,A -85,B 0,C 180,E1 14623.635,E2 14623.635} C_VEL
LIN {X 0,Y 336.671,Z 1223.896,A -85,B 0,C 180,E1 14620.35,E2 14620.35} C_VEL
LIN {X 0,Y 322.351,Z 1235.539,A -85,B 0,C 180,E1 14616.553,E2 14616.553} C_VEL
LIN {X 0,Y 310.292,Z 1245.27,A -85,B 0,C 180,E1 14612.403,E2 14612.403} C_VEL
LIN {X 0,Y 300.491,Z 1253.048,A -85,B 0,C 180,E1 14607.981,E2 14607.981} C_VEL
LIN {X 0,Y 292.695,Z 1259.053,A -85,B 0,C 180,E1 14603.223,E2 14603.223} C_VEL
LIN {X 0,Y 287.196,Z 1262.988,A -85,B 0,C 180,E1 14598.471,E2 14598.471} C_VEL
LIN {X 0,Y 283.679,Z 1265.075,A -85,B 0,C 180,E1 14593.868,E2 14593.868} C_VEL
LIN {X 0,Y 281.556,Z 1265.394,A -85,B 0,C 180,E1 14589.196,E2 14589.196} C_VEL
LIN {X 0,Y 280.563,Z 1264.086,A -85,B 0,C 180,E1 14584.702,E2 14584.702} C_VEL
LIN {X 0,Y 280.235,Z 1261.51,A -85,B 0,C 180,E1 14580.613,E2 14580.613} C_VEL
LIN {X 0,Y 280.163,Z 1257.557,A -85,B 0,C 180,E1 14576.726,E2 14576.726} C_VEL
LIN {X 0,Y 280.364,Z 1251.893,A -85,B 0,C 180,E1 14572.623,E2 14572.623} C_VEL
LIN {X 0,Y 280.895,Z 1245.26,A -85,B 0,C 180,E1 14568.917,E2 14568.917} C_VEL
LIN {X 0,Y 282.022,Z 1236.52,A -85,B 0,C 180,E1 14565,E2 14565} C_VEL
LIN {X 0,Y 283.87,Z 1225.894,A -85,B 0,C 180,E1 14561.091,E2 14561.091} C_VEL
LIN {X 0,Y 286.388,Z 1213.851,A -85,B 0,C 180,E1 14557.415,E2 14557.415} C_VEL
LIN {X 0,Y 289.708,Z 1199.493,A -85,B 0,C 180,E1 14553.783,E2 14553.783} C_VEL
LIN {X 0,Y 293.495,Z 1184.039,A -85,B 0,C 180,E1 14550.509,E2 14550.509} C_VEL
LIN {X 0,Y 297.822,Z 1166.74,A -85,B 0,C 180,E1 14547.429,E2 14547.429} C_VEL
LIN {X 0,Y 302.581,Z 1147.389,A -85,B 0,C 180,E1 14544.553,E2 14544.553} C_VEL
LIN {X 0,Y 307.335,Z 1127.13,A -85,B 0,C 180,E1 14542.055,E2 14542.055} C_VEL
LIN {X 0,Y 311.763,Z 1106.914,A -85,B 0,C 180,E1 14539.98,E2 14539.98} C_VEL
LIN {X 0,Y 316.258,Z 1084.402,A -85,B 0,C 180,E1 14538.086,E2 14538.086} C_VEL
LIN {X 0,Y 320.322,Z 1061.03,A -85,B 0,C 180,E1 14536.504,E2 14536.504} C_VEL
LIN {X 0,Y 324.001,Z 1035.92,A -85,B 0,C 180,E1 14535.188,E2 14535.188} C_VEL
LIN {X 0,Y 326.934,Z 1010.471,A -85,B 0,C 180,E1 14534.205,E2 14534.205} C_VEL
LIN {X 0,Y 346.835,Z 813.48,A -85,B 0,C 180,E1 14528.384,E2 14528.384} C_VEL
LIN {X 0,Y 332.544,Z 785.048,A -85,B 0,C 180,E1 14525.237,E2 14525.237} C_VEL
LIN {X 0,Y 319.17,Z 760.35,A -85,B 0,C 180,E1 14522.049,E2 14522.049} C_VEL
LIN {X 0,Y 306.563,Z 738.649,A -85,B 0,C 180,E1 14518.785,E2 14518.785} C_VEL
LIN {X 0,Y 294.393,Z 718.911,A -85,B 0,C 180,E1 14515.34,E2 14515.34} C_VEL
LIN {X 0,Y 292.273,Z 715.539,A -85,B 0,C 180,E1 14514.671,E2 14514.671} C_VEL
LIN {X 0,Y 287.333,Z 705.517,A -85,B 0,C 180,E1 14511.863,E2 14511.863} C_VEL
LIN {X 0,Y 285.412,Z 701.515,A -85,B 0,C 180,E1 14510.708,E2 14510.708} C_VEL
LIN {X 0,Y 283.8,Z 698.44,A -85,B 0,C 180,E1 14509.772,E2 14509.772} C_VEL
LIN {X 0,Y 283.58,Z 697.34,A -85,B 0,C 180,E1 14509.507,E2 14509.507} C_VEL
LIN {X 0,Y 283.586,Z 697.335,A -85,B 0,C 180,E1 14504.709,E2 14504.709} C_VEL
LIN {X 0,Y 283.576,Z 697.336,A -85,B 0,C 180,E1 14499.952,E2 14499.952} C_VEL
LIN {X 0,Y 283.579,Z 697.336,A -85,B 0,C 180,E1 14495.466,E2 14495.466} C_VEL
LIN {X 0,Y 283.596,Z 697.49,A -85,B 0,C 180,E1 14492.428,E2 14492.428} C_VEL
LIN {X 0,Y 285.006,Z 700.979,A -85,B 0,C 180,E1 14490.606,E2 14490.606} C_VEL
LIN {X 0,Y 286.423,Z 702.769,A -85,B 0,C 180,E1 14489.403,E2 14489.403} C_VEL
LIN {X 0,Y 288.25,Z 706.622,A -85,B 0,C 180,E1 14487.474,E2 14487.474} C_VEL
LIN {X 0,Y 289.193,Z 708.184,A -85,B 0,C 180,E1 14486.633,E2 14486.633} C_VEL
LIN {X 0,Y 291.752,Z 713.075,A -85,B 0,C 180,E1 14484.299,E2 14484.299} C_VEL
LIN {X 0,Y 294.342,Z 718.323,A -85,B 0,C 180,E1 14481.997,E2 14481.997} C_VEL
LIN {X 0,Y 296.871,Z 723.382,A -85,B 0,C 180,E1 14479.916,E2 14479.916} C_VEL
LIN {X 0,Y 300.477,Z 730.646,A -85,B 0,C 180,E1 14477.12,E2 14477.12} C_VEL
LIN {X 0,Y 305.658,Z 741.804,A -85,B 0,C 180,E1 14473.272,E2 14473.272} C_VEL
LIN {X 0,Y 311.48,Z 755.465,A -85,B 0,C 180,E1 14469.128,E2 14469.128} C_VEL
LIN {X 0,Y 316.95,Z 769.306,A -85,B 0,C 180,E1 14465.394,E2 14465.394} C_VEL
LIN {X 0,Y 322.483,Z 784.677,A -85,B 0,C 180,E1 14461.684,E2 14461.684} C_VEL
LIN {X 0,Y 328.182,Z 802.153,A -85,B 0,C 180,E1 14457.887,E2 14457.887} C_VEL
LIN {X 0,Y 332.01,Z 815.49,A -85,B 0,C 180,E1 14455.257,E2 14455.257} C_VEL
LIN {X 0,Y 322.544,Z 856.839,A -85,B 0,C 180,E1 14450.386,E2 14450.386} C_VEL
LIN {X 0,Y 313.582,Z 900.269,A -85,B 0,C 180,E1 14445.201,E2 14445.201} C_VEL
LIN {X 0,Y 308.601,Z 927.648,A -85,B 0,C 180,E1 14441.941,E2 14441.941} C_VEL
LIN {X 0,Y 308.592,Z 939.305,A -85,B 0,C 180,E1 14441.391,E2 14441.391} C_VEL
LIN {X 0,Y 302.291,Z 1004.012,A -85,B 0,C 180,E1 14438.709,E2 14438.709} C_VEL
LIN {X 0,Y 297.246,Z 1057.189,A -85,B 0,C 180,E1 14436.087,E2 14436.087} C_VEL
LIN {X 0,Y 295.089,Z 1085.138,A -85,B 0,C 180,E1 14434.463,E2 14434.463} C_VEL
LIN {X 0,Y 293.344,Z 1102.875,A -85,B 0,C 180,E1 14433.05,E2 14433.05} C_VEL
LIN {X 0,Y 291.248,Z 1120.409,A -85,B 0,C 180,E1 14431.225,E2 14431.225} C_VEL
LIN {X 0,Y 289.125,Z 1136.575,A -85,B 0,C 180,E1 14429.071,E2 14429.071} C_VEL
LIN {X 0,Y 287.118,Z 1150.814,A -85,B 0,C 180,E1 14426.695,E2 14426.695} C_VEL
LIN {X 0,Y 285.278,Z 1164.027,A -85,B 0,C 180,E1 14423.99,E2 14423.99} C_VEL
LIN {X 0,Y 284.363,Z 1170.973,A -85,B 0,C 180,E1 14422.303,E2 14422.303} C_VEL
LIN {X 0,Y 282.811,Z 1175.649,A -85,B 0,C 180,E1 14421.089,E2 14421.089} C_VEL
LIN {X 0,Y 277.161,Z 1184.019,A -85,B 0,C 180,E1 14418.633,E2 14418.633} C_VEL
LIN {X 0,Y 274.804,Z 1188.369,A -85,B 0,C 180,E1 14417.089,E2 14417.089} C_VEL
LIN {X 0,Y 274.493,Z 1189.923,A -85,B 0,C 180,E1 14416.475,E2 14416.475} C_VEL
LIN {X 0,Y 274.233,Z 1197.983,A -85,B 0,C 180,E1 14412.851,E2 14412.851} C_VEL
LIN {X 0,Y 274.599,Z 1203.989,A -85,B 0,C 180,E1 14409.219,E2 14409.219} C_VEL
LIN {X 0,Y 275.658,Z 1208.185,A -85,B 0,C 180,E1 14405.62,E2 14405.62} C_VEL
LIN {X 0,Y 277.784,Z 1210.861,A -85,B 0,C 180,E1 14401.65,E2 14401.65} C_VEL
LIN {X 0,Y 280.839,Z 1211.529,A -85,B 0,C 180,E1 14397.96,E2 14397.96} C_VEL
LIN {X 0,Y 284.966,Z 1210.487,A -85,B 0,C 180,E1 14394.362,E2 14394.362} C_VEL
LIN {X 0,Y 290.505,Z 1207.463,A -85,B 0,C 180,E1 14390.69,E2 14390.69} C_VEL
LIN {X 0,Y 296.868,Z 1202.781,A -85,B 0,C 180,E1 14387.354,E2 14387.354} C_VEL
LIN {X 0,Y 304.28,Z 1196.256,A -85,B 0,C 180,E1 14384.172,E2 14384.172} C_VEL
LIN {X 0,Y 312.716,Z 1187.688,A -85,B 0,C 180,E1 14381.159,E2 14381.159} C_VEL
LIN {X 0,Y 321.595,Z 1177.535,A -85,B 0,C 180,E1 14378.477,E2 14378.477} C_VEL
LIN {X 0,Y 331.364,Z 1165.066,A -85,B 0,C 180,E1 14375.961,E2 14375.961} C_VEL
LIN {X 0,Y 341.075,Z 1151.226,A -85,B 0,C 180,E1 14373.819,E2 14373.819} C_VEL
LIN {X 0,Y 350.863,Z 1135.571,A -85,B 0,C 180,E1 14371.951,E2 14371.951} C_VEL
LIN {X 0,Y 359.9,Z 1119.349,A -85,B 0,C 180,E1 14370.453,E2 14370.453} C_VEL
LIN {X 0,Y 371.641,Z 1096.189,A -85,B 0,C 180,E1 14368.817,E2 14368.817} C_VEL
LIN {X 0,Y 383.593,Z 1070.921,A -85,B 0,C 180,E1 14367.434,E2 14367.434} C_VEL
LIN {X 0,Y 395.503,Z 1042.63,A -85,B 0,C 180,E1 14366.207,E2 14366.207} C_VEL
LIN {X 0,Y 397.547,Z 1037.211,A -85,B 0,C 180,E1 14365.987,E2 14365.987} C_VEL
LIN {X 0,Y 389.25,Z 1059.132,A -85,B 0,C 180,E1 14365.281,E2 14365.281} C_VEL
LIN {X 0,Y 378.957,Z 1083.357,A -85,B 0,C 180,E1 14364.223,E2 14364.223} C_VEL
LIN {X 0,Y 367.916,Z 1106.849,A -85,B 0,C 180,E1 14362.901,E2 14362.901} C_VEL
LIN {X 0,Y 355.657,Z 1130.656,A -85,B 0,C 180,E1 14361.142,E2 14361.142} C_VEL
LIN {X 0,Y 344.178,Z 1150.804,A -85,B 0,C 180,E1 14359.206,E2 14359.206} C_VEL
LIN {X 0,Y 332.601,Z 1169.355,A -85,B 0,C 180,E1 14356.926,E2 14356.926} C_VEL
LIN {X 0,Y 321.101,Z 1186.631,A -85,B 0,C 180,E1 14354.224,E2 14354.224} C_VEL
LIN {X 0,Y 310.712,Z 1201.645,A -85,B 0,C 180,E1 14351.273,E2 14351.273} C_VEL
LIN {X 0,Y 301.023,Z 1215.443,A -85,B 0,C 180,E1 14347.912,E2 14347.912} C_VEL
LIN {X 0,Y 291.625,Z 1229.012,A -85,B 0,C 180,E1 14343.738,E2 14343.738} C_VEL
LIN {X 0,Y 283.837,Z 1240.79,A -85,B 0,C 180,E1 14339.084,E2 14339.084} C_VEL
LIN {X 0,Y 278.061,Z 1250.563,A -85,B 0,C 180,E1 14334.024,E2 14334.024} C_VEL
LIN {X 0,Y 274.631,Z 1257.888,A -85,B 0,C 180,E1 14328.904,E2 14328.904} C_VEL
LIN {X 0,Y 273.48,Z 1261.91,A -85,B 0,C 180,E1 14325.259,E2 14325.259} C_VEL
LIN {X 0,Y 272.797,Z 1270.158,A -85,B 0,C 180,E1 14321.413,E2 14321.413} C_VEL
LIN {X 0,Y 272.662,Z 1276.571,A -85,B 0,C 180,E1 14317.583,E2 14317.583} C_VEL
LIN {X 0,Y 272.744,Z 1281.49,A -85,B 0,C 180,E1 14313.781,E2 14313.781} C_VEL
LIN {X 0,Y 272.741,Z 1284.596,A -85,B 0,C 180,E1 14310.207,E2 14310.207} C_VEL
LIN {X 0,Y 272.493,Z 1286.408,A -85,B 0,C 180,E1 14306.842,E2 14306.842} C_VEL
LIN {X 0,Y 272.226,Z 1287.243,A -85,B 0,C 180,E1 14302.611,E2 14302.611} C_VEL
LIN {X 0,Y 272.494,Z 1286.553,A -85,B 0,C 180,E1 14298.354,E2 14298.354} C_VEL
LIN {X 0,Y 274.173,Z 1283.958,A -85,B 0,C 180,E1 14293.253,E2 14293.253} C_VEL
LIN {X 0,Y 277.684,Z 1279.578,A -85,B 0,C 180,E1 14288.227,E2 14288.227} C_VEL
LIN {X 0,Y 283.49,Z 1273.11,A -85,B 0,C 180,E1 14283.16,E2 14283.16} C_VEL
LIN {X 0,Y 291.584,Z 1264.838,A -85,B 0,C 180,E1 14278.352,E2 14278.352} C_VEL
LIN {X 0,Y 302.914,Z 1254.029,A -85,B 0,C 180,E1 14273.545,E2 14273.545} C_VEL
LIN {X 0,Y 316.817,Z 1241.422,A -85,B 0,C 180,E1 14269.207,E2 14269.207} C_VEL
LIN {X 0,Y 332.585,Z 1227.728,A -85,B 0,C 180,E1 14265.531,E2 14265.531} C_VEL
LIN {X 0,Y 342.957,Z 1218.894,A -85,B 0,C 180,E1 14263.564,E2 14263.564} C_VEL
LIN {X 0,Y 326.276,Z 1231.287,A -85,B 0,C 180,E1 14259.989,E2 14259.989} C_VEL
LIN {X 0,Y 311.787,Z 1241.932,A -85,B 0,C 180,E1 14255.936,E2 14255.936} C_VEL
LIN {X 0,Y 299.868,Z 1250.539,A -85,B 0,C 180,E1 14251.568,E2 14251.568} C_VEL
LIN {X 0,Y 290.499,Z 1257.09,A -85,B 0,C 180,E1 14247.023,E2 14247.023} C_VEL
LIN {X 0,Y 282.969,Z 1262.055,A -85,B 0,C 180,E1 14241.997,E2 14241.997} C_VEL
LIN {X 0,Y 277.981,Z 1264.916,A -85,B 0,C 180,E1 14237.155,E2 14237.155} C_VEL
LIN {X 0,Y 274.847,Z 1266.045,A -85,B 0,C 180,E1 14232.395,E2 14232.395} C_VEL
LIN {X 0,Y 273.15,Z 1265.463,A -85,B 0,C 180,E1 14227.784,E2 14227.784} C_VEL
LIN {X 0,Y 272.383,Z 1263.305,A -85,B 0,C 180,E1 14223.12,E2 14223.12} C_VEL
LIN {X 0,Y 272.191,Z 1260.115,A -85,B 0,C 180,E1 14219.158,E2 14219.158} C_VEL
LIN {X 0,Y 272.211,Z 1255.17,A -85,B 0,C 180,E1 14214.942,E2 14214.942} C_VEL
LIN {X 0,Y 272.549,Z 1248.982,A -85,B 0,C 180,E1 14210.923,E2 14210.923} C_VEL
LIN {X 0,Y 273.381,Z 1241.016,A -85,B 0,C 180,E1 14206.893,E2 14206.893} C_VEL
LIN {X 0,Y 274.891,Z 1231.221,A -85,B 0,C 180,E1 14202.865,E2 14202.865} C_VEL
LIN {X 0,Y 277.075,Z 1220.088,A -85,B 0,C 180,E1 14199.068,E2 14199.068} C_VEL
LIN {X 0,Y 280.067,Z 1206.882,A -85,B 0,C 180,E1 14195.31,E2 14195.31} C_VEL
LIN {X 0,Y 283.726,Z 1191.916,A -85,B 0,C 180,E1 14191.771,E2 14191.771} C_VEL
LIN {X 0,Y 287.795,Z 1175.89,A -85,B 0,C 180,E1 14188.591,E2 14188.591} C_VEL
LIN {X 0,Y 292.458,Z 1157.567,A -85,B 0,C 180,E1 14185.54,E2 14185.54} C_VEL
LIN {X 0,Y 297.407,Z 1137.469,A -85,B 0,C 180,E1 14182.759,E2 14182.759} C_VEL
LIN {X 0,Y 302.139,Z 1117.158,A -85,B 0,C 180,E1 14180.427,E2 14180.427} C_VEL
LIN {X 0,Y 306.658,Z 1096.162,A -85,B 0,C 180,E1 14178.43,E2 14178.43} C_VEL
LIN {X 0,Y 311.023,Z 1073.475,A -85,B 0,C 180,E1 14176.671,E2 14176.671} C_VEL
LIN {X 0,Y 314.994,Z 1049.438,A -85,B 0,C 180,E1 14175.194,E2 14175.194} C_VEL
LIN {X 0,Y 318.366,Z 1024.462,A -85,B 0,C 180,E1 14174.026,E2 14174.026} C_VEL
LIN {X 0,Y 322.33,Z 986.02,A -85,B 0,C 180,E1 14172.748,E2 14172.748} C_VEL
LIN {X 0,Y 340.247,Z 816.259,A -85,B 0,C 180,E1 14167.656,E2 14167.656} C_VEL
LIN {X 0,Y 326.14,Z 788.092,A -85,B 0,C 180,E1 14164.449,E2 14164.449} C_VEL
LIN {X 0,Y 312.922,Z 763.68,A -85,B 0,C 180,E1 14161.203,E2 14161.203} C_VEL
LIN {X 0,Y 300.211,Z 741.645,A -85,B 0,C 180,E1 14157.796,E2 14157.796} C_VEL
LIN {X 0,Y 287.119,Z 720.528,A -85,B 0,C 180,E1 14153.938,E2 14153.938} C_VEL
LIN {X 0,Y 284.253,Z 715.922,A -85,B 0,C 180,E1 14152.985,E2 14152.985} C_VEL
LIN {X 0,Y 279.275,Z 706.262,A -85,B 0,C 180,E1 14150.106,E2 14150.106} C_VEL
LIN {X 0,Y 277.387,Z 702.402,A -85,B 0,C 180,E1 14148.933,E2 14148.933} C_VEL
LIN {X 0,Y 275.814,Z 699.25,A -85,B 0,C 180,E1 14147.95,E2 14147.95} C_VEL
LIN {X 0,Y 275.641,Z 698.331,A -85,B 0,C 180,E1 14147.634,E2 14147.634} C_VEL
LIN {X 0,Y 275.644,Z 698.309,A -85,B 0,C 180,E1 14142.787,E2 14142.787} C_VEL
LIN {X 0,Y 275.65,Z 698.31,A -85,B 0,C 180,E1 14137.926,E2 14137.926} C_VEL
LIN {X 0,Y 275.658,Z 698.401,A -85,B 0,C 180,E1 14136.145,E2 14136.145} C_VEL
LIN {X 0,Y 276.961,Z 701.831,A -85,B 0,C 180,E1 14134.143,E2 14134.143} C_VEL
LIN {X 0,Y 278.537,Z 703.676,A -85,B 0,C 180,E1 14132.678,E2 14132.678} C_VEL
LIN {X 0,Y 280.215,Z 707.429,A -85,B 0,C 180,E1 14130.616,E2 14130.616} C_VEL
LIN {X 0,Y 281.332,Z 709,A -85,B 0,C 180,E1 14129.595,E2 14129.595} C_VEL
LIN {X 0,Y 283.262,Z 712.859,A -85,B 0,C 180,E1 14127.575,E2 14127.575} C_VEL
LIN {X 0,Y 284.455,Z 715.344,A -85,B 0,C 180,E1 14126.375,E2 14126.375} C_VEL
LIN {X 0,Y 286.441,Z 718.882,A -85,B 0,C 180,E1 14124.595,E2 14124.595} C_VEL
LIN {X 0,Y 289.235,Z 724.651,A -85,B 0,C 180,E1 14122.054,E2 14122.054} C_VEL
LIN {X 0,Y 292.764,Z 731.536,A -85,B 0,C 180,E1 14119.176,E2 14119.176} C_VEL
LIN {X 0,Y 298.266,Z 743.367,A -85,B 0,C 180,E1 14114.845,E2 14114.845} C_VEL
LIN {X 0,Y 303.955,Z 756.681,A -85,B 0,C 180,E1 14110.598,E2 14110.598} C_VEL
LIN {X 0,Y 309.605,Z 770.841,A -85,B 0,C 180,E1 14106.598,E2 14106.598} C_VEL
LIN {X 0,Y 315.062,Z 785.912,A -85,B 0,C 180,E1 14102.809,E2 14102.809} C_VEL
LIN {X 0,Y 320.543,Z 802.678,A -85,B 0,C 180,E1 14099.026,E2 14099.026} C_VEL
LIN {X 0,Y 325.055,Z 818.279,A -85,B 0,C 180,E1 14095.839,E2 14095.839} C_VEL
LIN {X 0,Y 315.267,Z 859.852,A -85,B 0,C 180,E1 14090.87,E2 14090.87} C_VEL
LIN {X 0,Y 305.834,Z 904.461,A -85,B 0,C 180,E1 14085.457,E2 14085.457} C_VEL
LIN {X 0,Y 301.353,Z 928.515,A -85,B 0,C 180,E1 14082.556,E2 14082.556} C_VEL
LIN {X 0,Y 301.327,Z 939.707,A -85,B 0,C 180,E1 14082.021,E2 14082.021} C_VEL
LIN {X 0,Y 295.35,Z 999.08,A -85,B 0,C 180,E1 14079.5,E2 14079.5} C_VEL
LIN {X 0,Y 289.813,Z 1054.919,A -85,B 0,C 180,E1 14076.688,E2 14076.688} C_VEL
LIN {X 0,Y 287.349,Z 1085.641,A -85,B 0,C 180,E1 14074.858,E2 14074.858} C_VEL
LIN {X 0,Y 285.575,Z 1103.258,A -85,B 0,C 180,E1 14073.425,E2 14073.425} C_VEL
LIN {X 0,Y 283.459,Z 1120.395,A -85,B 0,C 180,E1 14071.59,E2 14071.59} C_VEL
LIN {X 0,Y 281.357,Z 1135.987,A -85,B 0,C 180,E1 14069.469,E2 14069.469} C_VEL
LIN {X 0,Y 279.29,Z 1150.444,A -85,B 0,C 180,E1 14067.044,E2 14067.044} C_VEL
LIN {X 0,Y 277.353,Z 1164.108,A -85,B 0,C 180,E1 14064.213,E2 14064.213} C_VEL
LIN {X 0,Y 275.862,Z 1175.662,A -85,B 0,C 180,E1 14061.252,E2 14061.252} C_VEL
LIN {X 0,Y 274.803,Z 1185.845,A -85,B 0,C 180,E1 14058.016,E2 14058.016} C_VEL
LIN {X 0,Y 274.493,Z 1189.923,A -85,B 0,C 180,E1 14056.475,E2 14056.475} C_VEL
LIN {X 0,Y 273.317,Z 1193.402,A -85,B 0,C 180,E1 14055.041,E2 14055.041} C_VEL
LIN {X 0,Y 268.454,Z 1199.522,A -85,B 0,C 180,E1 14052.161,E2 14052.161} C_VEL
LIN {X 0,Y 266.616,Z 1202.564,A -85,B 0,C 180,E1 14050.407,E2 14050.407} C_VEL
LIN {X 0,Y 266.516,Z 1203.627,A -85,B 0,C 180,E1 14049.729,E2 14049.729} C_VEL
LIN {X 0,Y 267.503,Z 1208.298,A -85,B 0,C 180,E1 14046.008,E2 14046.008} C_VEL
LIN {X 0,Y 269.449,Z 1211.44,A -85,B 0,C 180,E1 14042.127,E2 14042.127} C_VEL
LIN {X 0,Y 272.629,Z 1212.734,A -85,B 0,C 180,E1 14038.108,E2 14038.108} C_VEL
LIN {X 0,Y 276.782,Z 1212.2,A -85,B 0,C 180,E1 14034.403,E2 14034.403} C_VEL
LIN {X 0,Y 282.397,Z 1209.791,A -85,B 0,C 180,E1 14030.626,E2 14030.626} C_VEL
LIN {X 0,Y 289.47,Z 1205.264,A -85,B 0,C 180,E1 14026.912,E2 14026.912} C_VEL
LIN {X 0,Y 297.307,Z 1199.057,A -85,B 0,C 180,E1 14023.59,E2 14023.59} C_VEL
LIN {X 0,Y 306.016,Z 1191.014,A -85,B 0,C 180,E1 14020.532,E2 14020.532} C_VEL
LIN {X 0,Y 315.458,Z 1181.146,A -85,B 0,C 180,E1 14017.741,E2 14017.741} C_VEL
LIN {X 0,Y 325.208,Z 1169.729,A -85,B 0,C 180,E1 14015.282,E2 14015.282} C_VEL
LIN {X 0,Y 335.072,Z 1156.886,A -85,B 0,C 180,E1 14013.15,E2 14013.15} C_VEL
LIN {X 0,Y 344.833,Z 1142.74,A -85,B 0,C 180,E1 14011.322,E2 14011.322} C_VEL
LIN {X 0,Y 354.399,Z 1127.252,A -85,B 0,C 180,E1 14009.76,E2 14009.76} C_VEL
LIN {X 0,Y 364.229,Z 1109.489,A -85,B 0,C 180,E1 14008.376,E2 14008.376} C_VEL
LIN {X 0,Y 376.103,Z 1086.635,A -85,B 0,C 180,E1 14006.975,E2 14006.975} C_VEL
LIN {X 0,Y 384.572,Z 1069.144,A -85,B 0,C 180,E1 14006.095,E2 14006.095} C_VEL
LIN {X 0,Y 372.776,Z 1094.694,A -85,B 0,C 180,E1 14004.89,E2 14004.89} C_VEL
LIN {X 0,Y 361.302,Z 1117.045,A -85,B 0,C 180,E1 14003.504,E2 14003.504} C_VEL
LIN {X 0,Y 350.786,Z 1136.021,A -85,B 0,C 180,E1 14002.007,E2 14002.007} C_VEL
LIN {X 0,Y 338.963,Z 1155.218,A -85,B 0,C 180,E1 14000.077,E2 14000.077} C_VEL
LIN {X 0,Y 326.842,Z 1173.209,A -85,B 0,C 180,E1 13997.756,E2 13997.756} C_VEL
LIN {X 0,Y 314.44,Z 1190.428,A -85,B 0,C 180,E1 13994.901,E2 13994.901} C_VEL
LIN {X 0,Y 302.734,Z 1206.023,A -85,B 0,C 180,E1 13991.592,E2 13991.592} C_VEL
LIN {X 0,Y 292.919,Z 1218.91,A -85,B 0,C 180,E1 13988.155,E2 13988.155} C_VEL
LIN {X 0,Y 283.788,Z 1231.082,A -85,B 0,C 180,E1 13984.067,E2 13984.067} C_VEL
LIN {X 0,Y 276.135,Z 1241.699,A -85,B 0,C 180,E1 13979.498,E2 13979.498} C_VEL
LIN {X 0,Y 270.725,Z 1249.998,A -85,B 0,C 180,E1 13974.897,E2 13974.897} C_VEL
LIN {X 0,Y 267.15,Z 1256.657,A -85,B 0,C 180,E1 13970.041,E2 13970.041} C_VEL
LIN {X 0,Y 265.461,Z 1261.658,A -85,B 0,C 180,E1 13965.061,E2 13965.061} C_VEL
LIN {X 0,Y 264.811,Z 1269.877,A -85,B 0,C 180,E1 13961.1,E2 13961.1} C_VEL
LIN {X 0,Y 264.72,Z 1276.223,A -85,B 0,C 180,E1 13957.157,E2 13957.157} C_VEL
LIN {X 0,Y 264.808,Z 1281.079,A -85,B 0,C 180,E1 13953.244,E2 13953.244} C_VEL
LIN {X 0,Y 264.759,Z 1284.124,A -85,B 0,C 180,E1 13949.564,E2 13949.564} C_VEL
LIN {X 0,Y 264.464,Z 1285.888,A -85,B 0,C 180,E1 13946.095,E2 13946.095} C_VEL
LIN {X 0,Y 264.234,Z 1286.681,A -85,B 0,C 180,E1 13941.51,E2 13941.51} C_VEL
LIN {X 0,Y 264.798,Z 1285.875,A -85,B 0,C 180,E1 13936.902,E2 13936.902} C_VEL
LIN {X 0,Y 267.001,Z 1283.158,A -85,B 0,C 180,E1 13931.662,E2 13931.662} C_VEL
LIN {X 0,Y 271.188,Z 1278.74,A -85,B 0,C 180,E1 13926.531,E2 13926.531} C_VEL
LIN {X 0,Y 278.137,Z 1272.057,A -85,B 0,C 180,E1 13921.199,E2 13921.199} C_VEL
LIN {X 0,Y 287.772,Z 1263.362,A -85,B 0,C 180,E1 13916.143,E2 13916.143} C_VEL
LIN {X 0,Y 300.661,Z 1252.378,A -85,B 0,C 180,E1 13911.299,E2 13911.299} C_VEL
LIN {X 0,Y 315.843,Z 1239.993,A -85,B 0,C 180,E1 13907.104,E2 13907.104} C_VEL
LIN {X 0,Y 333.12,Z 1226.383,A -85,B 0,C 180,E1 13903.481,E2 13903.481} C_VEL
LIN {X 0,Y 316.185,Z 1237.771,A -85,B 0,C 180,E1 13899.702,E2 13899.702} C_VEL
LIN {X 0,Y 301.679,Z 1247.339,A -85,B 0,C 180,E1 13895.452,E2 13895.452} C_VEL
LIN {X 0,Y 289.962,Z 1254.836,A -85,B 0,C 180,E1 13890.918,E2 13890.918} C_VEL
LIN {X 0,Y 280.528,Z 1260.565,A -85,B 0,C 180,E1 13886.003,E2 13886.003} C_VEL
LIN {X 0,Y 273.405,Z 1264.441,A -85,B 0,C 180,E1 13880.778,E2 13880.778} C_VEL
LIN {X 0,Y 268.848,Z 1266.329,A -85,B 0,C 180,E1 13875.754,E2 13875.754} C_VEL
LIN {X 0,Y 266.124,Z 1266.485,A -85,B 0,C 180,E1 13870.828,E2 13870.828} C_VEL
LIN {X 0,Y 264.772,Z 1265.004,A -85,B 0,C 180,E1 13866.07,E2 13866.07} C_VEL
LIN {X 0,Y 264.275,Z 1262.13,A -85,B 0,C 180,E1 13861.518,E2 13861.518} C_VEL
LIN {X 0,Y 264.164,Z 1258.327,A -85,B 0,C 180,E1 13857.614,E2 13857.614} C_VEL
LIN {X 0,Y 264.308,Z 1252.609,A -85,B 0,C 180,E1 13853.265,E2 13853.265} C_VEL
LIN {X 0,Y 264.844,Z 1245.553,A -85,B 0,C 180,E1 13849.119,E2 13849.119} C_VEL
LIN {X 0,Y 265.992,Z 1236.652,A -85,B 0,C 180,E1 13844.967,E2 13844.967} C_VEL
LIN {X 0,Y 267.954,Z 1225.641,A -85,B 0,C 180,E1 13840.756,E2 13840.756} C_VEL
LIN {X 0,Y 270.56,Z 1213.636,A -85,B 0,C 180,E1 13836.937,E2 13836.937} C_VEL
LIN {X 0,Y 274.065,Z 1199.154,A -85,B 0,C 180,E1 13833.102,E2 13833.102} C_VEL
LIN {X 0,Y 278.206,Z 1182.977,A -85,B 0,C 180,E1 13829.551,E2 13829.551} C_VEL
LIN {X 0,Y 282.697,Z 1165.753,A -85,B 0,C 180,E1 13826.39,E2 13826.39} C_VEL
LIN {X 0,Y 287.512,Z 1146.999,A -85,B 0,C 180,E1 13823.509,E2 13823.509} C_VEL
LIN {X 0,Y 292.544,Z 1126.467,A -85,B 0,C 180,E1 13820.887,E2 13820.887} C_VEL
LIN {X 0,Y 297.384,Z 1105.265,A -85,B 0,C 180,E1 13818.651,E2 13818.651} C_VEL
LIN {X 0,Y 301.995,Z 1082.98,A -85,B 0,C 180,E1 13816.735,E2 13816.735} C_VEL
LIN {X 0,Y 306.211,Z 1059.635,A -85,B 0,C 180,E1 13815.122,E2 13815.122} C_VEL
LIN {X 0,Y 309.888,Z 1035.582,A -85,B 0,C 180,E1 13813.825,E2 13813.825} C_VEL
LIN {X 0,Y 312.931,Z 1010.5,A -85,B 0,C 180,E1 13812.818,E2 13812.818} C_VEL
LIN {X 0,Y 333.577,Z 818.847,A -85,B 0,C 180,E1 13806.896,E2 13806.896} C_VEL
LIN {X 0,Y 319.935,Z 791.515,A -85,B 0,C 180,E1 13803.695,E2 13803.695} C_VEL
LIN {X 0,Y 306.542,Z 766.697,A -85,B 0,C 180,E1 13800.291,E2 13800.291} C_VEL
LIN {X 0,Y 294.214,Z 745.386,A -85,B 0,C 180,E1 13796.875,E2 13796.875} C_VEL
LIN {X 0,Y 282.31,Z 726.075,A -85,B 0,C 180,E1 13793.263,E2 13793.263} C_VEL
LIN {X 0,Y 276.181,Z 716.558,A -85,B 0,C 180,E1 13791.228,E2 13791.228} C_VEL
LIN {X 0,Y 271.62,Z 707.648,A -85,B 0,C 180,E1 13788.459,E2 13788.459} C_VEL
LIN {X 0,Y 269.787,Z 703.784,A -85,B 0,C 180,E1 13787.25,E2 13787.25} C_VEL
LIN {X 0,Y 268.083,Z 700.956,A -85,B 0,C 180,E1 13786.247,E2 13786.247} C_VEL
LIN {X 0,Y 267.703,Z 699.321,A -85,B 0,C 180,E1 13785.77,E2 13785.77} C_VEL
LIN {X 0,Y 267.705,Z 699.319,A -85,B 0,C 180,E1 13780.984,E2 13780.984} C_VEL
LIN {X 0,Y 267.714,Z 699.401,A -85,B 0,C 180,E1 13780.548,E2 13780.548} C_VEL
LIN {X 0,Y 269.249,Z 703.11,A -85,B 0,C 180,E1 13777.9,E2 13777.9} C_VEL
LIN {X 0,Y 270.802,Z 705.141,A -85,B 0,C 180,E1 13776.15,E2 13776.15} C_VEL
LIN {X 0,Y 272.588,Z 708.798,A -85,B 0,C 180,E1 13773.789,E2 13773.789} C_VEL
LIN {X 0,Y 273.604,Z 710.275,A -85,B 0,C 180,E1 13772.726,E2 13772.726} C_VEL
LIN {X 0,Y 275.65,Z 714.145,A -85,B 0,C 180,E1 13770.418,E2 13770.418} C_VEL
LIN {X 0,Y 278.818,Z 720.211,A -85,B 0,C 180,E1 13767.125,E2 13767.125} C_VEL
LIN {X 0,Y 281.513,Z 725.642,A -85,B 0,C 180,E1 13764.5,E2 13764.5} C_VEL
LIN {X 0,Y 283.923,Z 730.497,A -85,B 0,C 180,E1 13762.312,E2 13762.312} C_VEL
LIN {X 0,Y 287.382,Z 737.444,A -85,B 0,C 180,E1 13759.377,E2 13759.377} C_VEL
LIN {X 0,Y 292.619,Z 748.818,A -85,B 0,C 180,E1 13755.154,E2 13755.154} C_VEL
LIN {X 0,Y 298.247,Z 762.192,A -85,B 0,C 180,E1 13750.822,E2 13750.822} C_VEL
LIN {X 0,Y 303.563,Z 775.787,A -85,B 0,C 180,E1 13746.926,E2 13746.926} C_VEL
LIN {X 0,Y 308.945,Z 790.932,A -85,B 0,C 180,E1 13743.06,E2 13743.06} C_VEL
LIN {X 0,Y 314.095,Z 806.983,A -85,B 0,C 180,E1 13739.383,E2 13739.383} C_VEL
LIN {X 0,Y 318.122,Z 821.132,A -85,B 0,C 180,E1 13736.44,E2 13736.44} C_VEL
LIN {X 0,Y 307.946,Z 863.151,A -85,B 0,C 180,E1 13731.343,E2 13731.343} C_VEL
LIN {X 0,Y 298.468,Z 906.615,A -85,B 0,C 180,E1 13725.975,E2 13725.975} C_VEL
LIN {X 0,Y 294.134,Z 929.177,A -85,B 0,C 180,E1 13723.209,E2 13723.209} C_VEL
LIN {X 0,Y 294.043,Z 940.256,A -85,B 0,C 180,E1 13722.659,E2 13722.659} C_VEL
LIN {X 0,Y 287.539,Z 1002.781,A -85,B 0,C 180,E1 13719.91,E2 13719.91} C_VEL
LIN {X 0,Y 281.998,Z 1057.519,A -85,B 0,C 180,E1 13717.045,E2 13717.045} C_VEL
LIN {X 0,Y 279.573,Z 1086.469,A -85,B 0,C 180,E1 13715.237,E2 13715.237} C_VEL
LIN {X 0,Y 277.703,Z 1104.22,A -85,B 0,C 180,E1 13713.729,E2 13713.729} C_VEL
LIN {X 0,Y 275.453,Z 1121.954,A -85,B 0,C 180,E1 13711.759,E2 13711.759} C_VEL
LIN {X 0,Y 273.227,Z 1137.992,A -85,B 0,C 180,E1 13709.486,E2 13709.486} C_VEL
LIN {X 0,Y 271.139,Z 1152.309,A -85,B 0,C 180,E1 13706.975,E2 13706.975} C_VEL
LIN {X 0,Y 269.235,Z 1165.564,A -85,B 0,C 180,E1 13704.112,E2 13704.112} C_VEL
LIN {X 0,Y 267.646,Z 1177.864,A -85,B 0,C 180,E1 13700.788,E2 13700.788} C_VEL
LIN {X 0,Y 266.672,Z 1187.777,A -85,B 0,C 180,E1 13697.455,E2 13697.455} C_VEL
LIN {X 0,Y 266.25,Z 1196.209,A -85,B 0,C 180,E1 13693.907,E2 13693.907} C_VEL
LIN {X 0,Y 266.419,Z 1202.612,A -85,B 0,C 180,E1 13690.378,E2 13690.378} C_VEL
LIN {X 0,Y 266.516,Z 1203.627,A -85,B 0,C 180,E1 13689.729,E2 13689.729} C_VEL
LIN {X 0,Y 265.857,Z 1206.001,A -85,B 0,C 180,E1 13688.143,E2 13688.143} C_VEL
LIN {X 0,Y 262.032,Z 1209.968,A -85,B 0,C 180,E1 13684.826,E2 13684.826} C_VEL
LIN {X 0,Y 261.094,Z 1211.581,A -85,B 0,C 180,E1 13682.913,E2 13682.913} C_VEL
LIN {X 0,Y 261.302,Z 1211.983,A -85,B 0,C 180,E1 13682.311,E2 13682.311} C_VEL
LIN {X 0,Y 264.405,Z 1213.812,A -85,B 0,C 180,E1 13678.266,E2 13678.266} C_VEL
LIN {X 0,Y 268.845,Z 1213.725,A -85,B 0,C 180,E1 13674.237,E2 13674.237} C_VEL
LIN {X 0,Y 274.256,Z 1211.943,A -85,B 0,C 180,E1 13670.557,E2 13670.557} C_VEL
LIN {X 0,Y 281.46,Z 1208.077,A -85,B 0,C 180,E1 13666.736,E2 13666.736} C_VEL
LIN {X 0,Y 289.89,Z 1202.177,A -85,B 0,C 180,E1 13663.158,E2 13663.158} C_VEL
LIN {X 0,Y 299.024,Z 1194.577,A -85,B 0,C 180,E1 13659.978,E2 13659.978} C_VEL
LIN {X 0,Y 308.194,Z 1185.899,A -85,B 0,C 180,E1 13657.289,E2 13657.289} C_VEL
LIN {X 0,Y 317.835,Z 1175.729,A -85,B 0,C 180,E1 13654.868,E2 13654.868} C_VEL
LIN {X 0,Y 328.298,Z 1163.438,A -85,B 0,C 180,E1 13652.619,E2 13652.619} C_VEL
LIN {X 0,Y 339.206,Z 1149.094,A -85,B 0,C 180,E1 13650.607,E2 13650.607} C_VEL
LIN {X 0,Y 350.132,Z 1132.995,A -85,B 0,C 180,E1 13648.876,E2 13648.876} C_VEL
LIN {X 0,Y 361.423,Z 1114.103,A -85,B 0,C 180,E1 13647.352,E2 13647.352} C_VEL
LIN {X 0,Y 372.017,Z 1095.012,A -85,B 0,C 180,E1 13646.147,E2 13646.147} C_VEL
LIN {X 0,Y 359.856,Z 1117.896,A -85,B 0,C 180,E1 13644.771,E2 13644.771} C_VEL
LIN {X 0,Y 348.252,Z 1137.683,A -85,B 0,C 180,E1 13643.226,E2 13643.226} C_VEL
LIN {X 0,Y 336.768,Z 1155.265,A -85,B 0,C 180,E1 13641.472,E2 13641.472} C_VEL
LIN {X 0,Y 325.174,Z 1171.568,A -85,B 0,C 180,E1 13639.416,E2 13639.416} C_VEL
LIN {X 0,Y 312.105,Z 1188.659,A -85,B 0,C 180,E1 13636.651,E2 13636.651} C_VEL
LIN {X 0,Y 299.655,Z 1204.131,A -85,B 0,C 180,E1 13633.419,E2 13633.419} C_VEL
LIN {X 0,Y 289.104,Z 1216.939,A -85,B 0,C 180,E1 13630.034,E2 13630.034} C_VEL
LIN {X 0,Y 278.977,Z 1229.274,A -85,B 0,C 180,E1 13625.902,E2 13625.902} C_VEL
LIN {X 0,Y 270.293,Z 1240.151,A -85,B 0,C 180,E1 13621.187,E2 13621.187} C_VEL
LIN {X 0,Y 263.974,Z 1248.753,A -85,B 0,C 180,E1 13616.303,E2 13616.303} C_VEL
LIN {X 0,Y 259.762,Z 1255.488,A -85,B 0,C 180,E1 13611.209,E2 13611.209} C_VEL
LIN {X 0,Y 257.582,Z 1260.562,A -85,B 0,C 180,E1 13605.699,E2 13605.699} C_VEL
LIN {X 0,Y 257.447,Z 1261.367,A -85,B 0,C 180,E1 13604.849,E2 13604.849} C_VEL
LIN {X 0,Y 256.836,Z 1269.535,A -85,B 0,C 180,E1 13600.767,E2 13600.767} C_VEL
LIN {X 0,Y 256.792,Z 1275.839,A -85,B 0,C 180,E1 13596.705,E2 13596.705} C_VEL
LIN {X 0,Y 256.88,Z 1280.631,A -85,B 0,C 180,E1 13592.674,E2 13592.674} C_VEL
LIN {X 0,Y 256.77,Z 1283.623,A -85,B 0,C 180,E1 13588.881,E2 13588.881} C_VEL
LIN {X 0,Y 256.412,Z 1285.422,A -85,B 0,C 180,E1 13585.076,E2 13585.076} C_VEL
LIN {X 0,Y 256.292,Z 1286.107,A -85,B 0,C 180,E1 13580.34,E2 13580.34} C_VEL
LIN {X 0,Y 257.24,Z 1285.192,A -85,B 0,C 180,E1 13575.362,E2 13575.362} C_VEL
LIN {X 0,Y 260.034,Z 1282.393,A -85,B 0,C 180,E1 13569.985,E2 13569.985} C_VEL
LIN {X 0,Y 265.469,Z 1277.503,A -85,B 0,C 180,E1 13564.33,E2 13564.33} C_VEL
LIN {X 0,Y 273.53,Z 1270.797,A -85,B 0,C 180,E1 13558.971,E2 13558.971} C_VEL
LIN {X 0,Y 284.646,Z 1261.923,A -85,B 0,C 180,E1 13553.83,E2 13553.83} C_VEL
LIN {X 0,Y 298.46,Z 1251.371,A -85,B 0,C 180,E1 13549.208,E2 13549.208} C_VEL
LIN {X 0,Y 314.803,Z 1239.34,A -85,B 0,C 180,E1 13545.158,E2 13545.158} C_VEL
LIN {X 0,Y 323.317,Z 1233.208,A -85,B 0,C 180,E1 13543.419,E2 13543.419} C_VEL
LIN {X 0,Y 306.434,Z 1243.432,A -85,B 0,C 180,E1 13539.515,E2 13539.515} C_VEL
LIN {X 0,Y 292.027,Z 1251.904,A -85,B 0,C 180,E1 13535.116,E2 13535.116} C_VEL
LIN {X 0,Y 280.441,Z 1258.404,A -85,B 0,C 180,E1 13530.417,E2 13530.417} C_VEL
LIN {X 0,Y 270.898,Z 1263.337,A -85,B 0,C 180,E1 13525.117,E2 13525.117} C_VEL
LIN {X 0,Y 264.355,Z 1266.165,A -85,B 0,C 180,E1 13519.902,E2 13519.902} C_VEL
LIN {X 0,Y 260.092,Z 1267.224,A -85,B 0,C 180,E1 13514.698,E2 13514.698} C_VEL
LIN {X 0,Y 257.659,Z 1266.514,A -85,B 0,C 180,E1 13509.606,E2 13509.606} C_VEL
LIN {X 0,Y 256.554,Z 1264.303,A -85,B 0,C 180,E1 13504.695,E2 13504.695} C_VEL
LIN {X 0,Y 256.227,Z 1261.068,A -85,B 0,C 180,E1 13500.447,E2 13500.447} C_VEL
LIN {X 0,Y 256.174,Z 1256.429,A -85,B 0,C 180,E1 13496.195,E2 13496.195} C_VEL
LIN {X 0,Y 256.437,Z 1250.348,A -85,B 0,C 180,E1 13491.931,E2 13491.931} C_VEL
LIN {X 0,Y 257.159,Z 1242.499,A -85,B 0,C 180,E1 13487.652,E2 13487.652} C_VEL
LIN {X 0,Y 258.592,Z 1232.872,A -85,B 0,C 180,E1 13483.373,E2 13483.373} C_VEL
LIN {X 0,Y 260.74,Z 1221.939,A -85,B 0,C 180,E1 13479.341,E2 13479.341} C_VEL
LIN {X 0,Y 263.752,Z 1208.822,A -85,B 0,C 180,E1 13475.354,E2 13475.354} C_VEL
LIN {X 0,Y 267.429,Z 1194.258,A -85,B 0,C 180,E1 13471.651,E2 13471.651} C_VEL
LIN {X 0,Y 271.803,Z 1177.757,A -85,B 0,C 180,E1 13468.136,E2 13468.136} C_VEL
LIN {X 0,Y 276.625,Z 1159.666,A -85,B 0,C 180,E1 13464.92,E2 13464.92} C_VEL
LIN {X 0,Y 281.579,Z 1140.589,A -85,B 0,C 180,E1 13462.097,E2 13462.097} C_VEL
LIN {X 0,Y 286.681,Z 1119.862,A -85,B 0,C 180,E1 13459.554,E2 13459.554} C_VEL
LIN {X 0,Y 291.595,Z 1098.249,A -85,B 0,C 180,E1 13457.372,E2 13457.372} C_VEL
LIN {X 0,Y 296.403,Z 1074.515,A -85,B 0,C 180,E1 13455.438,E2 13455.438} C_VEL
LIN {X 0,Y 300.649,Z 1050.163,A -85,B 0,C 180,E1 13453.874,E2 13453.874} C_VEL
LIN {X 0,Y 304.289,Z 1024.691,A -85,B 0,C 180,E1 13452.626,E2 13452.626} C_VEL
LIN {X 0,Y 308.873,Z 982.792,A -85,B 0,C 180,E1 13451.17,E2 13451.17} C_VEL
LIN {X 0,Y 327.005,Z 821.582,A -85,B 0,C 180,E1 13446.12,E2 13446.12} C_VEL
LIN {X 0,Y 313.74,Z 794.94,A -85,B 0,C 180,E1 13442.917,E2 13442.917} C_VEL
LIN {X 0,Y 300.869,Z 770.976,A -85,B 0,C 180,E1 13439.547,E2 13439.547} C_VEL
LIN {X 0,Y 288.087,Z 748.693,A -85,B 0,C 180,E1 13435.88,E2 13435.88} C_VEL
LIN {X 0,Y 276.639,Z 730.306,A -85,B 0,C 180,E1 13432.287,E2 13432.287} C_VEL
LIN {X 0,Y 268.151,Z 717.22,A -85,B 0,C 180,E1 13429.373,E2 13429.373} C_VEL
LIN {X 0,Y 264.011,Z 709.065,A -85,B 0,C 180,E1 13426.731,E2 13426.731} C_VEL
LIN {X 0,Y 261.849,Z 704.776,A -85,B 0,C 180,E1 13425.28,E2 13425.28} C_VEL
LIN {X 0,Y 260.38,Z 702.528,A -85,B 0,C 180,E1 13424.344,E2 13424.344} C_VEL
LIN {X 0,Y 262.98,Z 706.197,A -85,B 0,C 180,E1 13420.518,E2 13420.518} C_VEL
LIN {X 0,Y 264.842,Z 709.967,A -85,B 0,C 180,E1 13417.596,E2 13417.596} C_VEL
LIN {X 0,Y 265.849,Z 711.239,A -85,B 0,C 180,E1 13416.482,E2 13416.482} C_VEL
LIN {X 0,Y 267.77,Z 715.181,A -85,B 0,C 180,E1 13413.857,E2 13413.857} C_VEL
LIN {X 0,Y 268.595,Z 716.424,A -85,B 0,C 180,E1 13412.99,E2 13412.99} C_VEL
LIN {X 0,Y 270.85,Z 720.569,A -85,B 0,C 180,E1 13410.426,E2 13410.426} C_VEL
LIN {X 0,Y 273.901,Z 726.881,A -85,B 0,C 180,E1 13407.073,E2 13407.073} C_VEL
LIN {X 0,Y 276.228,Z 731.456,A -85,B 0,C 180,E1 13404.811,E2 13404.811} C_VEL
LIN {X 0,Y 279.998,Z 738.995,A -85,B 0,C 180,E1 13401.377,E2 13401.377} C_VEL
LIN {X 0,Y 285.282,Z 750.446,A -85,B 0,C 180,E1 13396.834,E2 13396.834} C_VEL
LIN {X 0,Y 290.535,Z 762.859,A -85,B 0,C 180,E1 13392.581,E2 13392.581} C_VEL
LIN {X 0,Y 295.738,Z 776.021,A -85,B 0,C 180,E1 13388.587,E2 13388.587} C_VEL
LIN {X 0,Y 301.059,Z 790.655,A -85,B 0,C 180,E1 13384.635,E2 13384.635} C_VEL
LIN {X 0,Y 306.37,Z 807.086,A -85,B 0,C 180,E1 13380.692,E2 13380.692} C_VEL
LIN {X 0,Y 310.912,Z 822.726,A -85,B 0,C 180,E1 13377.3,E2 13377.3} C_VEL
LIN {X 0,Y 311.104,Z 824.252,A -85,B 0,C 180,E1 13377.02,E2 13377.02} C_VEL
LIN {X 0,Y 300.455,Z 867.031,A -85,B 0,C 180,E1 13371.757,E2 13371.757} C_VEL
LIN {X 0,Y 290.706,Z 910.746,A -85,B 0,C 180,E1 13366.268,E2 13366.268} C_VEL
LIN {X 0,Y 286.905,Z 929.865,A -85,B 0,C 180,E1 13363.872,E2 13363.872} C_VEL
LIN {X 0,Y 286.765,Z 940.799,A -85,B 0,C 180,E1 13363.317,E2 13363.317} C_VEL
LIN {X 0,Y 280.2,Z 1002.211,A -85,B 0,C 180,E1 13360.552,E2 13360.552} C_VEL
LIN {X 0,Y 274.824,Z 1052.766,A -85,B 0,C 180,E1 13357.835,E2 13357.835} C_VEL
LIN {X 0,Y 271.825,Z 1086.835,A -85,B 0,C 180,E1 13355.651,E2 13355.651} C_VEL
LIN {X 0,Y 269.943,Z 1104.295,A -85,B 0,C 180,E1 13354.137,E2 13354.137} C_VEL
LIN {X 0,Y 267.681,Z 1121.753,A -85,B 0,C 180,E1 13352.161,E2 13352.161} C_VEL
LIN {X 0,Y 265.505,Z 1137.203,A -85,B 0,C 180,E1 13349.952,E2 13349.952} C_VEL
LIN {X 0,Y 263.281,Z 1152.09,A -85,B 0,C 180,E1 13347.3,E2 13347.3} C_VEL
LIN {X 0,Y 261.213,Z 1166.157,A -85,B 0,C 180,E1 13344.179,E2 13344.179} C_VEL
LIN {X 0,Y 259.693,Z 1177.791,A -85,B 0,C 180,E1 13340.982,E2 13340.982} C_VEL
LIN {X 0,Y 258.685,Z 1187.959,A -85,B 0,C 180,E1 13337.547,E2 13337.547} C_VEL
LIN {X 0,Y 258.251,Z 1196.486,A -85,B 0,C 180,E1 13333.89,E2 13333.89} C_VEL
LIN {X 0,Y 258.441,Z 1203.118,A -85,B 0,C 180,E1 13330.252,E2 13330.252} C_VEL
LIN {X 0,Y 259.447,Z 1208.615,A -85,B 0,C 180,E1 13326.151,E2 13326.151} C_VEL
LIN {X 0,Y 261.302,Z 1211.983,A -85,B 0,C 180,E1 13322.311,E2 13322.311} C_VEL
LIN {X 0,Y 261.433,Z 1213.055,A -85,B 0,C 180,E1 13320.624,E2 13320.624} C_VEL
LIN {X 0,Y 259.328,Z 1215.047,A -85,B 0,C 180,E1 13316.24,E2 13316.24} C_VEL
LIN {X 0,Y 260.287,Z 1215.213,A -85,B 0,C 180,E1 13314.543,E2 13314.543} C_VEL
LIN {X 0,Y 265.752,Z 1214.052,A -85,B 0,C 180,E1 13310.689,E2 13310.689} C_VEL
LIN {X 0,Y 272.764,Z 1211.062,A -85,B 0,C 180,E1 13306.863,E2 13306.863} C_VEL
LIN {X 0,Y 281.518,Z 1205.839,A -85,B 0,C 180,E1 13303.067,E2 13303.067} C_VEL
LIN {X 0,Y 291.626,Z 1198.414,A -85,B 0,C 180,E1 13299.529,E2 13299.529} C_VEL
LIN {X 0,Y 302.425,Z 1189.137,A -85,B 0,C 180,E1 13296.418,E2 13296.418} C_VEL
LIN {X 0,Y 313.679,Z 1178.119,A -85,B 0,C 180,E1 13293.699,E2 13293.699} C_VEL
LIN {X 0,Y 325.256,Z 1165.36,A -85,B 0,C 180,E1 13291.343,E2 13291.343} C_VEL
LIN {X 0,Y 336.998,Z 1150.844,A -85,B 0,C 180,E1 13289.314,E2 13289.314} C_VEL
LIN {X 0,Y 347.941,Z 1135.623,A -85,B 0,C 180,E1 13287.689,E2 13287.689} C_VEL
LIN {X 0,Y 358.752,Z 1118.707,A -85,B 0,C 180,E1 13286.314,E2 13286.314} C_VEL
LIN {X 0,Y 359.852,Z 1116.914,A -85,B 0,C 180,E1 13286.176,E2 13286.176} C_VEL
LIN {X 0,Y 347.717,Z 1136.882,A -85,B 0,C 180,E1 13284.69,E2 13284.69} C_VEL
LIN {X 0,Y 334.837,Z 1155.606,A -85,B 0,C 180,E1 13282.869,E2 13282.869} C_VEL
LIN {X 0,Y 322.438,Z 1171.957,A -85,B 0,C 180,E1 13280.823,E2 13280.823} C_VEL
LIN {X 0,Y 309.484,Z 1187.873,A -85,B 0,C 180,E1 13278.268,E2 13278.268} C_VEL
LIN {X 0,Y 296.359,Z 1203.126,A -85,B 0,C 180,E1 13275.11,E2 13275.11} C_VEL
LIN {X 0,Y 284.223,Z 1216.753,A -85,B 0,C 180,E1 13271.467,E2 13271.467} C_VEL
LIN {X 0,Y 273.953,Z 1228.208,A -85,B 0,C 180,E1 13267.551,E2 13267.551} C_VEL
LIN {X 0,Y 264.38,Z 1239.101,A -85,B 0,C 180,E1 13262.736,E2 13262.736} C_VEL
LIN {X 0,Y 256.883,Z 1248.226,A -85,B 0,C 180,E1 13257.338,E2 13257.338} C_VEL
LIN {X 0,Y 252.104,Z 1254.932,A -85,B 0,C 180,E1 13251.886,E2 13251.886} C_VEL
LIN {X 0,Y 249.752,Z 1259.508,A -85,B 0,C 180,E1 13246.511,E2 13246.511} C_VEL
LIN {X 0,Y 249.458,Z 1260.856,A -85,B 0,C 180,E1 13244.708,E2 13244.708} C_VEL
LIN {X 0,Y 248.871,Z 1269.151,A -85,B 0,C 180,E1 13240.413,E2 13240.413} C_VEL
LIN {X 0,Y 248.868,Z 1275.418,A -85,B 0,C 180,E1 13236.224,E2 13236.224} C_VEL
LIN {X 0,Y 248.949,Z 1279.934,A -85,B 0,C 180,E1 13232.299,E2 13232.299} C_VEL
LIN {X 0,Y 248.785,Z 1282.955,A -85,B 0,C 180,E1 13228.385,E2 13228.385} C_VEL
LIN {X 0,Y 248.408,Z 1284.77,A -85,B 0,C 180,E1 13224.453,E2 13224.453} C_VEL
LIN {X 0,Y 248.367,Z 1285.555,A -85,B 0,C 180,E1 13219.559,E2 13219.559} C_VEL
LIN {X 0,Y 249.554,Z 1284.704,A -85,B 0,C 180,E1 13214.425,E2 13214.425} C_VEL
LIN {X 0,Y 252.93,Z 1281.954,A -85,B 0,C 180,E1 13208.67,E2 13208.67} C_VEL
LIN {X 0,Y 258.738,Z 1277.488,A -85,B 0,C 180,E1 13203.116,E2 13203.116} C_VEL
LIN {X 0,Y 267.821,Z 1270.761,A -85,B 0,C 180,E1 13197.476,E2 13197.476} C_VEL
LIN {X 0,Y 279.761,Z 1262.26,A -85,B 0,C 180,E1 13192.323,E2 13192.323} C_VEL
LIN {X 0,Y 295.577,Z 1251.402,A -85,B 0,C 180,E1 13187.421,E2 13187.421} C_VEL
LIN {X 0,Y 313.446,Z 1239.482,A -85,B 0,C 180,E1 13183.366,E2 13183.366} C_VEL
LIN {X 0,Y 296.639,Z 1248.589,A -85,B 0,C 180,E1 13179.324,E2 13179.324} C_VEL
LIN {X 0,Y 282.096,Z 1256.137,A -85,B 0,C 180,E1 13174.678,E2 13174.678} C_VEL
LIN {X 0,Y 270.501,Z 1261.738,A -85,B 0,C 180,E1 13169.691,E2 13169.691} C_VEL
LIN {X 0,Y 261.581,Z 1265.538,A -85,B 0,C 180,E1 13164.383,E2 13164.383} C_VEL
LIN {X 0,Y 255.322,Z 1267.52,A -85,B 0,C 180,E1 13158.968,E2 13158.968} C_VEL
LIN {X 0,Y 251.36,Z 1267.664,A -85,B 0,C 180,E1 13153.574,E2 13153.574} C_VEL
LIN {X 0,Y 249.256,Z 1266.19,A -85,B 0,C 180,E1 13148.303,E2 13148.303} C_VEL
LIN {X 0,Y 248.408,Z 1263.425,A -85,B 0,C 180,E1 13143.462,E2 13143.462} C_VEL
LIN {X 0,Y 248.193,Z 1259.47,A -85,B 0,C 180,E1 13139.077,E2 13139.077} C_VEL
LIN {X 0,Y 248.23,Z 1254.2,A -85,B 0,C 180,E1 13134.684,E2 13134.684} C_VEL
LIN {X 0,Y 248.613,Z 1247.675,A -85,B 0,C 180,E1 13130.509,E2 13130.509} C_VEL
LIN {X 0,Y 249.655,Z 1238.635,A -85,B 0,C 180,E1 13125.859,E2 13125.859} C_VEL
LIN {X 0,Y 251.345,Z 1228.748,A -85,B 0,C 180,E1 13121.683,E2 13121.683} C_VEL
LIN {X 0,Y 253.887,Z 1216.833,A -85,B 0,C 180,E1 13117.541,E2 13117.541} C_VEL
LIN {X 0,Y 257.127,Z 1203.583,A -85,B 0,C 180,E1 13113.684,E2 13113.684} C_VEL
LIN {X 0,Y 261.247,Z 1188.023,A -85,B 0,C 180,E1 13109.885,E2 13109.885} C_VEL
LIN {X 0,Y 265.86,Z 1171.082,A -85,B 0,C 180,E1 13106.436,E2 13106.436} C_VEL
LIN {X 0,Y 270.779,Z 1152.955,A -85,B 0,C 180,E1 13103.352,E2 13103.352} C_VEL
LIN {X 0,Y 276.221,Z 1132.125,A -85,B 0,C 180,E1 13100.424,E2 13100.424} C_VEL
LIN {X 0,Y 281.417,Z 1110.745,A -85,B 0,C 180,E1 13097.955,E2 13097.955} C_VEL
LIN {X 0,Y 286.404,Z 1088.369,A -85,B 0,C 180,E1 13095.853,E2 13095.853} C_VEL
LIN {X 0,Y 290.842,Z 1065.704,A -85,B 0,C 180,E1 13094.138,E2 13094.138} C_VEL
LIN {X 0,Y 294.808,Z 1041.923,A -85,B 0,C 180,E1 13092.716,E2 13092.716} C_VEL
LIN {X 0,Y 298.168,Z 1017.527,A -85,B 0,C 180,E1 13091.616,E2 13091.616} C_VEL
LIN {X 0,Y 320.385,Z 824.225,A -85,B 0,C 180,E1 13085.329,E2 13085.329} C_VEL
LIN {X 0,Y 307.333,Z 797.884,A -85,B 0,C 180,E1 13082.056,E2 13082.056} C_VEL
LIN {X 0,Y 294.361,Z 773.71,A -85,B 0,C 180,E1 13078.536,E2 13078.536} C_VEL
LIN {X 0,Y 282.615,Z 753.244,A -85,B 0,C 180,E1 13075.056,E2 13075.056} C_VEL
LIN {X 0,Y 271.609,Z 735.36,A -85,B 0,C 180,E1 13071.49,E2 13071.49} C_VEL
LIN {X 0,Y 263.153,Z 722.338,A -85,B 0,C 180,E1 13068.501,E2 13068.501} C_VEL
LIN {X 0,Y 259.896,Z 717.384,A -85,B 0,C 180,E1 13067.235,E2 13067.235} C_VEL
LIN {X 0,Y 256.103,Z 710.047,A -85,B 0,C 180,E1 13064.704,E2 13064.704} C_VEL
LIN {X 0,Y 255.621,Z 709.283,A -85,B 0,C 180,E1 13064.385,E2 13064.385} C_VEL
LIN {X 0,Y 258.072,Z 712.209,A -85,B 0,C 180,E1 13060.947,E2 13060.947} C_VEL
LIN {X 0,Y 260.028,Z 716.324,A -85,B 0,C 180,E1 13057.738,E2 13057.738} C_VEL
LIN {X 0,Y 260.968,Z 717.703,A -85,B 0,C 180,E1 13056.603,E2 13056.603} C_VEL
LIN {X 0,Y 263.2,Z 721.836,A -85,B 0,C 180,E1 13053.706,E2 13053.706} C_VEL
LIN {X 0,Y 266.269,Z 727.978,A -85,B 0,C 180,E1 13050.003,E2 13050.003} C_VEL
LIN {X 0,Y 268.649,Z 732.657,A -85,B 0,C 180,E1 13047.443,E2 13047.443} C_VEL
LIN {X 0,Y 271.094,Z 737.677,A -85,B 0,C 180,E1 13044.924,E2 13044.924} C_VEL
LIN {X 0,Y 274.625,Z 744.835,A -85,B 0,C 180,E1 13041.629,E2 13041.629} C_VEL
LIN {X 0,Y 279.866,Z 756.418,A -85,B 0,C 180,E1 13036.995,E2 13036.995} C_VEL
LIN {X 0,Y 284.841,Z 768.328,A -85,B 0,C 180,E1 13032.853,E2 13032.853} C_VEL
LIN {X 0,Y 290.242,Z 782.228,A -85,B 0,C 180,E1 13028.585,E2 13028.585} C_VEL
LIN {X 0,Y 295.469,Z 797.134,A -85,B 0,C 180,E1 13024.55,E2 13024.55} C_VEL
LIN {X 0,Y 300.533,Z 813.272,A -85,B 0,C 180,E1 13020.656,E2 13020.656} C_VEL
LIN {X 0,Y 304.246,Z 826.895,A -85,B 0,C 180,E1 13017.688,E2 13017.688} C_VEL
LIN {X 0,Y 293.395,Z 869.131,A -85,B 0,C 180,E1 13012.412,E2 13012.412} C_VEL
LIN {X 0,Y 283.466,Z 912.254,A -85,B 0,C 180,E1 13006.901,E2 13006.901} C_VEL
LIN {X 0,Y 279.715,Z 930.714,A -85,B 0,C 180,E1 13004.56,E2 13004.56} C_VEL
LIN {X 0,Y 279.516,Z 941.453,A -85,B 0,C 180,E1 13004.003,E2 13004.003} C_VEL
LIN {X 0,Y 273.196,Z 998.85,A -85,B 0,C 180,E1 13001.36,E2 13001.36} C_VEL
LIN {X 0,Y 267.161,Z 1053.48,A -85,B 0,C 180,E1 12998.324,E2 12998.324} C_VEL
LIN {X 0,Y 263.997,Z 1088.134,A -85,B 0,C 180,E1 12996.016,E2 12996.016} C_VEL
LIN {X 0,Y 261.986,Z 1106.071,A -85,B 0,C 180,E1 12994.392,E2 12994.392} C_VEL
LIN {X 0,Y 259.684,Z 1123.199,A -85,B 0,C 180,E1 12992.358,E2 12992.358} C_VEL
LIN {X 0,Y 257.356,Z 1139.084,A -85,B 0,C 180,E1 12989.964,E2 12989.964} C_VEL
LIN {X 0,Y 255.165,Z 1153.47,A -85,B 0,C 180,E1 12987.289,E2 12987.289} C_VEL
LIN {X 0,Y 253.059,Z 1167.688,A -85,B 0,C 180,E1 12984.015,E2 12984.015} C_VEL
LIN {X 0,Y 251.567,Z 1179.211,A -85,B 0,C 180,E1 12980.717,E2 12980.717} C_VEL
LIN {X 0,Y 250.604,Z 1189.21,A -85,B 0,C 180,E1 12977.173,E2 12977.173} C_VEL
LIN {X 0,Y 250.243,Z 1198.179,A -85,B 0,C 180,E1 12973.165,E2 12973.165} C_VEL
LIN {X 0,Y 250.617,Z 1204.999,A -85,B 0,C 180,E1 12969.183,E2 12969.183} C_VEL
LIN {X 0,Y 251.884,Z 1210.207,A -85,B 0,C 180,E1 12965.01,E2 12965.01} C_VEL
LIN {X 0,Y 254.349,Z 1213.667,A -85,B 0,C 180,E1 12960.676,E2 12960.676} C_VEL
LIN {X 0,Y 257.873,Z 1215.123,A -85,B 0,C 180,E1 12956.666,E2 12956.666} C_VEL
LIN {X 0,Y 260.287,Z 1215.213,A -85,B 0,C 180,E1 12954.543,E2 12954.543} C_VEL
LIN {X 0,Y 261.54,Z 1215.222,A -85,B 0,C 180,E1 12952.735,E2 12952.735} C_VEL
LIN {X 0,Y 262.234,Z 1214.709,A -85,B 0,C 180,E1 12948.58,E2 12948.58} C_VEL
LIN {X 0,Y 264.111,Z 1213.714,A -85,B 0,C 180,E1 12946.959,E2 12946.959} C_VEL
LIN {X 0,Y 264.321,Z 1213.616,A -85,B 0,C 180,E1 12946.85,E2 12946.85} C_VEL
LIN {X 0,Y 273.103,Z 1209.223,A -85,B 0,C 180,E1 12942.968,E2 12942.968} C_VEL
LIN {X 0,Y 283.327,Z 1202.679,A -85,B 0,C 180,E1 12939.334,E2 12939.334} C_VEL
LIN {X 0,Y 294.873,Z 1193.86,A -85,B 0,C 180,E1 12935.989,E2 12935.989} C_VEL
LIN {X 0,Y 306.327,Z 1183.785,A -85,B 0,C 180,E1 12933.227,E2 12933.227} C_VEL
LIN {X 0,Y 318.798,Z 1171.343,A -85,B 0,C 180,E1 12930.706,E2 12930.706} C_VEL
LIN {X 0,Y 330.739,Z 1157.958,A -85,B 0,C 180,E1 12928.668,E2 12928.668} C_VEL
LIN {X 0,Y 342.663,Z 1142.919,A -85,B 0,C 180,E1 12926.93,E2 12926.93} C_VEL
LIN {X 0,Y 348.03,Z 1135.553,A -85,B 0,C 180,E1 12926.205,E2 12926.205} C_VEL
LIN {X 0,Y 335.098,Z 1153.635,A -85,B 0,C 180,E1 12924.542,E2 12924.542} C_VEL
LIN {X 0,Y 322.165,Z 1169.926,A -85,B 0,C 180,E1 12922.606,E2 12922.606} C_VEL
LIN {X 0,Y 309.252,Z 1185.001,A -85,B 0,C 180,E1 12920.305,E2 12920.305} C_VEL
LIN {X 0,Y 295.271,Z 1200.266,A -85,B 0,C 180,E1 12917.288,E2 12917.288} C_VEL
LIN {X 0,Y 282.624,Z 1213.498,A -85,B 0,C 180,E1 12913.897,E2 12913.897} C_VEL
LIN {X 0,Y 270.341,Z 1226.095,A -85,B 0,C 180,E1 12909.707,E2 12909.707} C_VEL
LIN {X 0,Y 259.475,Z 1237.29,A -85,B 0,C 180,E1 12904.768,E2 12904.768} C_VEL
LIN {X 0,Y 250.994,Z 1246.411,A -85,B 0,C 180,E1 12899.336,E2 12899.336} C_VEL
LIN {X 0,Y 245.535,Z 1252.946,A -85,B 0,C 180,E1 12894.027,E2 12894.027} C_VEL
LIN {X 0,Y 242.358,Z 1257.731,A -85,B 0,C 180,E1 12888.519,E2 12888.519} C_VEL
LIN {X 0,Y 241.489,Z 1260.144,A -85,B 0,C 180,E1 12884.626,E2 12884.626} C_VEL
LIN {X 0,Y 240.938,Z 1268.082,A -85,B 0,C 180,E1 12880.406,E2 12880.406} C_VEL
LIN {X 0,Y 240.939,Z 1274.333,A -85,B 0,C 180,E1 12876.191,E2 12876.191} C_VEL
LIN {X 0,Y 241.027,Z 1278.45,A -85,B 0,C 180,E1 12872.612,E2 12872.612} C_VEL
LIN {X 0,Y 240.888,Z 1281.676,A -85,B 0,C 180,E1 12868.808,E2 12868.808} C_VEL
LIN {X 0,Y 240.443,Z 1283.945,A -85,B 0,C 180,E1 12864.269,E2 12864.269} C_VEL
LIN {X 0,Y 240.381,Z 1284.889,A -85,B 0,C 180,E1 12859.693,E2 12859.693} C_VEL
LIN {X 0,Y 241.728,Z 1284.349,A -85,B 0,C 180,E1 12853.907,E2 12853.907} C_VEL
LIN {X 0,Y 245.362,Z 1281.988,A -85,B 0,C 180,E1 12847.978,E2 12847.978} C_VEL
LIN {X 0,Y 251.827,Z 1277.624,A -85,B 0,C 180,E1 12842.058,E2 12842.058} C_VEL
LIN {X 0,Y 261.492,Z 1271.307,A -85,B 0,C 180,E1 12836.324,E2 12836.324} C_VEL
LIN {X 0,Y 274.588,Z 1263.026,A -85,B 0,C 180,E1 12830.95,E2 12830.95} C_VEL
LIN {X 0,Y 290.565,Z 1253.17,A -85,B 0,C 180,E1 12826.234,E2 12826.234} C_VEL
LIN {X 0,Y 303.363,Z 1245.3,A -85,B 0,C 180,E1 12823.281,E2 12823.281} C_VEL
LIN {X 0,Y 286.216,Z 1253.541,A -85,B 0,C 180,E1 12818.964,E2 12818.964} C_VEL
LIN {X 0,Y 271.635,Z 1260.104,A -85,B 0,C 180,E1 12814.022,E2 12814.022} C_VEL
LIN {X 0,Y 260.183,Z 1264.717,A -85,B 0,C 180,E1 12808.71,E2 12808.71} C_VEL
LIN {X 0,Y 251.708,Z 1267.476,A -85,B 0,C 180,E1 12803.158,E2 12803.158} C_VEL
LIN {X 0,Y 245.94,Z 1268.453,A -85,B 0,C 180,E1 12797.509,E2 12797.509} C_VEL
LIN {X 0,Y 242.486,Z 1267.62,A -85,B 0,C 180,E1 12791.898,E2 12791.898} C_VEL
LIN {X 0,Y 240.821,Z 1265.208,A -85,B 0,C 180,E1 12786.437,E2 12786.437} C_VEL
LIN {X 0,Y 240.285,Z 1261.743,A -85,B 0,C 180,E1 12781.669,E2 12781.669} C_VEL
LIN {X 0,Y 240.176,Z 1256.976,A -85,B 0,C 180,E1 12777.133,E2 12777.133} C_VEL
LIN {X 0,Y 240.377,Z 1250.838,A -85,B 0,C 180,E1 12772.591,E2 12772.591} C_VEL
LIN {X 0,Y 241.06,Z 1242.908,A -85,B 0,C 180,E1 12768.03,E2 12768.03} C_VEL
LIN {X 0,Y 242.492,Z 1233.185,A -85,B 0,C 180,E1 12763.47,E2 12763.47} C_VEL
LIN {X 0,Y 244.698,Z 1222.133,A -85,B 0,C 180,E1 12759.176,E2 12759.176} C_VEL
LIN {X 0,Y 247.829,Z 1208.98,A -85,B 0,C 180,E1 12754.936,E2 12754.936} C_VEL
LIN {X 0,Y 251.682,Z 1194.292,A -85,B 0,C 180,E1 12751.008,E2 12751.008} C_VEL
LIN {X 0,Y 256.279,Z 1177.659,A -85,B 0,C 180,E1 12747.291,E2 12747.291} C_VEL
LIN {X 0,Y 261.356,Z 1159.421,A -85,B 0,C 180,E1 12743.902,E2 12743.902} C_VEL
LIN {X 0,Y 266.573,Z 1140.228,A -85,B 0,C 180,E1 12740.938,E2 12740.938} C_VEL
LIN {X 0,Y 271.746,Z 1120.189,A -85,B 0,C 180,E1 12738.37,E2 12738.37} C_VEL
LIN {X 0,Y 276.875,Z 1098.676,A -85,B 0,C 180,E1 12736.102,E2 12736.102} C_VEL
LIN {X 0,Y 281.909,Z 1075.012,A -85,B 0,C 180,E1 12734.091,E2 12734.091} C_VEL
LIN {X 0,Y 286.486,Z 1050.003,A -85,B 0,C 180,E1 12732.421,E2 12732.421} C_VEL
LIN {X 0,Y 290.306,Z 1024.484,A -85,B 0,C 180,E1 12731.127,E2 12731.127} C_VEL
LIN {X 0,Y 296.71,Z 969.144,A -85,B 0,C 180,E1 12729.131,E2 12729.131} C_VEL
LIN {X 0,Y 313.789,Z 826.853,A -85,B 0,C 180,E1 12724.502,E2 12724.502} C_VEL
LIN {X 0,Y 301.121,Z 801.269,A -85,B 0,C 180,E1 12721.229,E2 12721.229} C_VEL
LIN {X 0,Y 288.543,Z 777.669,A -85,B 0,C 180,E1 12717.699,E2 12717.699} C_VEL
LIN {X 0,Y 277.008,Z 757.466,A -85,B 0,C 180,E1 12714.16,E2 12714.16} C_VEL
LIN {X 0,Y 265.767,Z 739.044,A -85,B 0,C 180,E1 12710.368,E2 12710.368} C_VEL
LIN {X 0,Y 256.11,Z 724.26,A -85,B 0,C 180,E1 12706.795,E2 12706.795} C_VEL
LIN {X 0,Y 251.746,Z 717.572,A -85,B 0,C 180,E1 12704.964,E2 12704.964} C_VEL
LIN {X 0,Y 250.951,Z 715.981,A -85,B 0,C 180,E1 12704.364,E2 12704.364} C_VEL
LIN {X 0,Y 252.129,Z 717.284,A -85,B 0,C 180,E1 12702.686,E2 12702.686} C_VEL
LIN {X 0,Y 253.328,Z 718.928,A -85,B 0,C 180,E1 12700.924,E2 12700.924} C_VEL
LIN {X 0,Y 255.442,Z 722.938,A -85,B 0,C 180,E1 12697.651,E2 12697.651} C_VEL
LIN {X 0,Y 256.349,Z 724.887,A -85,B 0,C 180,E1 12696.273,E2 12696.273} C_VEL
LIN {X 0,Y 258.652,Z 729.047,A -85,B 0,C 180,E1 12693.327,E2 12693.327} C_VEL
LIN {X 0,Y 261.062,Z 733.713,A -85,B 0,C 180,E1 12690.442,E2 12690.442} C_VEL
LIN {X 0,Y 263.753,Z 739.277,A -85,B 0,C 180,E1 12687.396,E2 12687.396} C_VEL
LIN {X 0,Y 267.149,Z 745.993,A -85,B 0,C 180,E1 12683.987,E2 12683.987} C_VEL
LIN {X 0,Y 272.169,Z 757.099,A -85,B 0,C 180,E1 12679.204,E2 12679.204} C_VEL
LIN {X 0,Y 277.009,Z 768.45,A -85,B 0,C 180,E1 12674.94,E2 12674.94} C_VEL
LIN {X 0,Y 282.016,Z 781.208,A -85,B 0,C 180,E1 12670.751,E2 12670.751} C_VEL
LIN {X 0,Y 287.14,Z 795.463,A -85,B 0,C 180,E1 12666.614,E2 12666.614} C_VEL
LIN {X 0,Y 292.051,Z 810.673,A -85,B 0,C 180,E1 12662.695,E2 12662.695} C_VEL
LIN {X 0,Y 296.886,Z 827.51,A -85,B 0,C 180,E1 12658.811,E2 12658.811} C_VEL
LIN {X 0,Y 297.264,Z 829.968,A -85,B 0,C 180,E1 12658.321,E2 12658.321} C_VEL
LIN {X 0,Y 286.173,Z 871.962,A -85,B 0,C 180,E1 12653.001,E2 12653.001} C_VEL
LIN {X 0,Y 276.102,Z 914.434,A -85,B 0,C 180,E1 12647.474,E2 12647.474} C_VEL
LIN {X 0,Y 272.531,Z 931.335,A -85,B 0,C 180,E1 12645.281,E2 12645.281} C_VEL
LIN {X 0,Y 272.298,Z 941.906,A -85,B 0,C 180,E1 12644.721,E2 12644.721} C_VEL
LIN {X 0,Y 265.603,Z 1000.599,A -85,B 0,C 180,E1 12641.921,E2 12641.921} C_VEL
LIN {X 0,Y 259.564,Z 1053.676,A -85,B 0,C 180,E1 12638.871,E2 12638.871} C_VEL
LIN {X 0,Y 256.264,Z 1088.509,A -85,B 0,C 180,E1 12636.468,E2 12636.468} C_VEL
LIN {X 0,Y 254.173,Z 1106.443,A -85,B 0,C 180,E1 12634.779,E2 12634.779} C_VEL
LIN {X 0,Y 251.723,Z 1124.185,A -85,B 0,C 180,E1 12632.599,E2 12632.599} C_VEL
LIN {X 0,Y 249.411,Z 1139.6,A -85,B 0,C 180,E1 12630.207,E2 12630.207} C_VEL
LIN {X 0,Y 247.095,Z 1154.556,A -85,B 0,C 180,E1 12627.341,E2 12627.341} C_VEL
LIN {X 0,Y 245.167,Z 1167.286,A -85,B 0,C 180,E1 12624.326,E2 12624.326} C_VEL
LIN {X 0,Y 243.613,Z 1178.997,A -85,B 0,C 180,E1 12620.921,E2 12620.921} C_VEL
LIN {X 0,Y 242.567,Z 1189.879,A -85,B 0,C 180,E1 12617.009,E2 12617.009} C_VEL
LIN {X 0,Y 242.247,Z 1198.906,A -85,B 0,C 180,E1 12612.879,E2 12612.879} C_VEL
LIN {X 0,Y 242.695,Z 1205.788,A -85,B 0,C 180,E1 12608.768,E2 12608.768} C_VEL
LIN {X 0,Y 244.099,Z 1211.129,A -85,B 0,C 180,E1 12604.464,E2 12604.464} C_VEL
LIN {X 0,Y 246.777,Z 1214.695,A -85,B 0,C 180,E1 12600,E2 12600} C_VEL
LIN {X 0,Y 250.617,Z 1216.331,A -85,B 0,C 180,E1 12595.833,E2 12595.833} C_VEL
LIN {X 0,Y 256.242,Z 1216.171,A -85,B 0,C 180,E1 12591.473,E2 12591.473} C_VEL
LIN {X 0,Y 263.459,Z 1213.971,A -85,B 0,C 180,E1 12587.284,E2 12587.284} C_VEL
LIN {X 0,Y 264.321,Z 1213.616,A -85,B 0,C 180,E1 12586.85,E2 12586.85} C_VEL
LIN {X 0,Y 266.709,Z 1212.377,A -85,B 0,C 180,E1 12585.15,E2 12585.15} C_VEL
LIN {X 0,Y 270.357,Z 1209.533,A -85,B 0,C 180,E1 12581.097,E2 12581.097} C_VEL
LIN {X 0,Y 272.834,Z 1207.924,A -85,B 0,C 180,E1 12579.845,E2 12579.845} C_VEL
LIN {X 0,Y 273.372,Z 1207.593,A -85,B 0,C 180,E1 12579.655,E2 12579.655} C_VEL
LIN {X 0,Y 283.636,Z 1200.956,A -85,B 0,C 180,E1 12576.525,E2 12576.525} C_VEL
LIN {X 0,Y 295.618,Z 1191.888,A -85,B 0,C 180,E1 12573.482,E2 12573.482} C_VEL
LIN {X 0,Y 307.993,Z 1181.163,A -85,B 0,C 180,E1 12570.858,E2 12570.858} C_VEL
LIN {X 0,Y 320.611,Z 1168.809,A -85,B 0,C 180,E1 12568.612,E2 12568.612} C_VEL
LIN {X 0,Y 333.3,Z 1154.8,A -85,B 0,C 180,E1 12566.702,E2 12566.702} C_VEL
LIN {X 0,Y 336.353,Z 1151.192,A -85,B 0,C 180,E1 12566.261,E2 12566.261} C_VEL
LIN {X 0,Y 323.079,Z 1167.271,A -85,B 0,C 180,E1 12564.478,E2 12564.478} C_VEL
LIN {X 0,Y 309.521,Z 1182.371,A -85,B 0,C 180,E1 12562.317,E2 12562.317} C_VEL
LIN {X 0,Y 295.404,Z 1196.935,A -85,B 0,C 180,E1 12559.599,E2 12559.599} C_VEL
LIN {X 0,Y 281.821,Z 1210.286,A -85,B 0,C 180,E1 12556.363,E2 12556.363} C_VEL
LIN {X 0,Y 267.992,Z 1223.37,A -85,B 0,C 180,E1 12552.185,E2 12552.185} C_VEL
LIN {X 0,Y 255.813,Z 1234.732,A -85,B 0,C 180,E1 12547.285,E2 12547.285} C_VEL
LIN {X 0,Y 246.786,Z 1243.334,A -85,B 0,C 180,E1 12542.327,E2 12542.327} C_VEL
LIN {X 0,Y 239.799,Z 1250.498,A -85,B 0,C 180,E1 12536.761,E2 12536.761} C_VEL
LIN {X 0,Y 235.134,Z 1256.106,A -85,B 0,C 180,E1 12530.404,E2 12530.404} C_VEL
LIN {X 0,Y 233.543,Z 1259.214,A -85,B 0,C 180,E1 12524.625,E2 12524.625} C_VEL
LIN {X 0,Y 233.01,Z 1266.998,A -85,B 0,C 180,E1 12520.38,E2 12520.38} C_VEL
LIN {X 0,Y 233.023,Z 1273.523,A -85,B 0,C 180,E1 12515.908,E2 12515.908} C_VEL
LIN {X 0,Y 233.113,Z 1277.668,A -85,B 0,C 180,E1 12512.209,E2 12512.209} C_VEL
LIN {X 0,Y 232.943,Z 1280.721,A -85,B 0,C 180,E1 12508.521,E2 12508.521} C_VEL
LIN {X 0,Y 232.456,Z 1283.182,A -85,B 0,C 180,E1 12503.823,E2 12503.823} C_VEL
LIN {X 0,Y 232.508,Z 1284.256,A -85,B 0,C 180,E1 12498.669,E2 12498.669} C_VEL
LIN {X 0,Y 234.253,Z 1283.805,A -85,B 0,C 180,E1 12492.612,E2 12492.612} C_VEL
LIN {X 0,Y 238.471,Z 1281.556,A -85,B 0,C 180,E1 12486.523,E2 12486.523} C_VEL
LIN {X 0,Y 245.665,Z 1277.376,A -85,B 0,C 180,E1 12480.493,E2 12480.493} C_VEL
LIN {X 0,Y 256.605,Z 1271.122,A -85,B 0,C 180,E1 12474.505,E2 12474.505} C_VEL
LIN {X 0,Y 270.7,Z 1263.221,A -85,B 0,C 180,E1 12469.169,E2 12469.169} C_VEL
LIN {X 0,Y 287.596,Z 1253.723,A -85,B 0,C 180,E1 12464.54,E2 12464.54} C_VEL
LIN {X 0,Y 293.388,Z 1250.508,A -85,B 0,C 180,E1 12463.238,E2 12463.238} C_VEL
LIN {X 0,Y 276.322,Z 1257.703,A -85,B 0,C 180,E1 12458.757,E2 12458.757} C_VEL
LIN {X 0,Y 261.87,Z 1263.258,A -85,B 0,C 180,E1 12453.618,E2 12453.618} C_VEL
LIN {X 0,Y 250.625,Z 1266.943,A -85,B 0,C 180,E1 12448.085,E2 12448.085} C_VEL
LIN {X 0,Y 242.432,Z 1268.827,A -85,B 0,C 180,E1 12442.3,E2 12442.3} C_VEL
LIN {X 0,Y 237.012,Z 1268.869,A -85,B 0,C 180,E1 12436.419,E2 12436.419} C_VEL
LIN {X 0,Y 233.93,Z 1267.238,A -85,B 0,C 180,E1 12430.591,E2 12430.591} C_VEL
LIN {X 0,Y 232.611,Z 1264.241,A -85,B 0,C 180,E1 12425.179,E2 12425.179} C_VEL
LIN {X 0,Y 232.241,Z 1260.259,A -85,B 0,C 180,E1 12420.493,E2 12420.493} C_VEL
LIN {X 0,Y 232.203,Z 1254.962,A -85,B 0,C 180,E1 12415.802,E2 12415.802} C_VEL
LIN {X 0,Y 232.514,Z 1248.44,A -85,B 0,C 180,E1 12411.343,E2 12411.343} C_VEL
LIN {X 0,Y 233.479,Z 1239.406,A -85,B 0,C 180,E1 12406.376,E2 12406.376} C_VEL
LIN {X 0,Y 235.143,Z 1229.511,A -85,B 0,C 180,E1 12401.916,E2 12401.916} C_VEL
LIN {X 0,Y 237.72,Z 1217.624,A -85,B 0,C 180,E1 12397.495,E2 12397.495} C_VEL
LIN {X 0,Y 241.054,Z 1204.37,A -85,B 0,C 180,E1 12393.385,E2 12393.385} C_VEL
LIN {X 0,Y 245.391,Z 1188.583,A -85,B 0,C 180,E1 12389.294,E2 12389.294} C_VEL
LIN {X 0,Y 250.137,Z 1171.918,A -85,B 0,C 180,E1 12385.693,E2 12385.693} C_VEL
LIN {X 0,Y 255.226,Z 1154.046,A -85,B 0,C 180,E1 12382.468,E2 12382.468} C_VEL
LIN {X 0,Y 260.969,Z 1133.073,A -85,B 0,C 180,E1 12379.357,E2 12379.357} C_VEL
LIN {X 0,Y 266.644,Z 1110.849,A -85,B 0,C 180,E1 12376.667,E2 12376.667} C_VEL
LIN {X 0,Y 272.042,Z 1087.728,A -85,B 0,C 180,E1 12374.41,E2 12374.41} C_VEL
LIN {X 0,Y 277.048,Z 1063.166,A -85,B 0,C 180,E1 12372.501,E2 12372.501} C_VEL
LIN {X 0,Y 281.372,Z 1038.035,A -85,B 0,C 180,E1 12370.991,E2 12370.991} C_VEL
LIN {X 0,Y 284.921,Z 1012.193,A -85,B 0,C 180,E1 12369.845,E2 12369.845} C_VEL
LIN {X 0,Y 307.203,Z 829.542,A -85,B 0,C 180,E1 12363.661,E2 12363.661} C_VEL
LIN {X 0,Y 294.443,Z 803.622,A -85,B 0,C 180,E1 12360.23,E2 12360.23} C_VEL
LIN {X 0,Y 281.605,Z 779.519,A -85,B 0,C 180,E1 12356.485,E2 12356.485} C_VEL
LIN {X 0,Y 269.745,Z 758.842,A -85,B 0,C 180,E1 12352.678,E2 12352.678} C_VEL
LIN {X 0,Y 258.736,Z 740.856,A -85,B 0,C 180,E1 12348.771,E2 12348.771} C_VEL
LIN {X 0,Y 249.247,Z 726.459,A -85,B 0,C 180,E1 12345.058,E2 12345.058} C_VEL
LIN {X 0,Y 246.71,Z 722.679,A -85,B 0,C 180,E1 12343.987,E2 12343.987} C_VEL
LIN {X 0,Y 248.536,Z 725.306,A -85,B 0,C 180,E1 12341.137,E2 12341.137} C_VEL
LIN {X 0,Y 250.85,Z 729.541,A -85,B 0,C 180,E1 12337.561,E2 12337.561} C_VEL
LIN {X 0,Y 253.636,Z 735.154,A -85,B 0,C 180,E1 12333.619,E2 12333.619} C_VEL
LIN {X 0,Y 256.174,Z 740.294,A -85,B 0,C 180,E1 12330.45,E2 12330.45} C_VEL
LIN {X 0,Y 258.658,Z 745.439,A -85,B 0,C 180,E1 12327.566,E2 12327.566} C_VEL
LIN {X 0,Y 261.977,Z 752.277,A -85,B 0,C 180,E1 12324.088,E2 12324.088} C_VEL
LIN {X 0,Y 266.773,Z 762.941,A -85,B 0,C 180,E1 12319.42,E2 12319.42} C_VEL
LIN {X 0,Y 271.549,Z 774.448,A -85,B 0,C 180,E1 12315.066,E2 12315.066} C_VEL
LIN {X 0,Y 276.497,Z 787.373,A -85,B 0,C 180,E1 12310.79,E2 12310.79} C_VEL
LIN {X 0,Y 281.559,Z 801.846,A -85,B 0,C 180,E1 12306.566,E2 12306.566} C_VEL
LIN {X 0,Y 286.383,Z 817.327,A -85,B 0,C 180,E1 12302.56,E2 12302.56} C_VEL
LIN {X 0,Y 290.507,Z 832.215,A -85,B 0,C 180,E1 12299.087,E2 12299.087} C_VEL
LIN {X 0,Y 279.33,Z 873.289,A -85,B 0,C 180,E1 12293.802,E2 12293.802} C_VEL
LIN {X 0,Y 268.888,Z 915.933,A -85,B 0,C 180,E1 12288.156,E2 12288.156} C_VEL
LIN {X 0,Y 265.37,Z 932.214,A -85,B 0,C 180,E1 12286.017,E2 12286.017} C_VEL
LIN {X 0,Y 265.063,Z 942.507,A -85,B 0,C 180,E1 12285.453,E2 12285.453} C_VEL
LIN {X 0,Y 258.066,Z 1002.054,A -85,B 0,C 180,E1 12282.528,E2 12282.528} C_VEL
LIN {X 0,Y 252.104,Z 1052.736,A -85,B 0,C 180,E1 12279.519,E2 12279.519} C_VEL
LIN {X 0,Y 248.422,Z 1089.625,A -85,B 0,C 180,E1 12276.85,E2 12276.85} C_VEL
LIN {X 0,Y 246.229,Z 1107.786,A -85,B 0,C 180,E1 12275.072,E2 12275.072} C_VEL
LIN {X 0,Y 243.7,Z 1125.615,A -85,B 0,C 180,E1 12272.792,E2 12272.792} C_VEL
LIN {X 0,Y 241.265,Z 1141.405,A -85,B 0,C 180,E1 12270.235,E2 12270.235} C_VEL
LIN {X 0,Y 239.022,Z 1155.506,A -85,B 0,C 180,E1 12267.397,E2 12267.397} C_VEL
LIN {X 0,Y 236.878,Z 1169.552,A -85,B 0,C 180,E1 12263.905,E2 12263.905} C_VEL
LIN {X 0,Y 235.401,Z 1181.012,A -85,B 0,C 180,E1 12260.384,E2 12260.384} C_VEL
LIN {X 0,Y 234.497,Z 1191.075,A -85,B 0,C 180,E1 12256.6,E2 12256.6} C_VEL
LIN {X 0,Y 234.266,Z 1200.218,A -85,B 0,C 180,E1 12252.221,E2 12252.221} C_VEL
LIN {X 0,Y 234.845,Z 1206.922,A -85,B 0,C 180,E1 12248.077,E2 12248.077} C_VEL
LIN {X 0,Y 236.453,Z 1212.249,A -85,B 0,C 180,E1 12243.637,E2 12243.637} C_VEL
LIN {X 0,Y 239.433,Z 1215.86,A -85,B 0,C 180,E1 12239.043,E2 12239.043} C_VEL
LIN {X 0,Y 243.57,Z 1217.558,A -85,B 0,C 180,E1 12234.818,E2 12234.818} C_VEL
LIN {X 0,Y 249.692,Z 1217.498,A -85,B 0,C 180,E1 12230.317,E2 12230.317} C_VEL
LIN {X 0,Y 257.697,Z 1215.324,A -85,B 0,C 180,E1 12225.92,E2 12225.92} C_VEL
LIN {X 0,Y 266.6,Z 1211.352,A -85,B 0,C 180,E1 12222.089,E2 12222.089} C_VEL
LIN {X 0,Y 273.372,Z 1207.593,A -85,B 0,C 180,E1 12219.655,E2 12219.655} C_VEL
LIN {X 0,Y 276.805,Z 1205.335,A -85,B 0,C 180,E1 12218.146,E2 12218.146} C_VEL
LIN {X 0,Y 283.03,Z 1200.455,A -85,B 0,C 180,E1 12214.493,E2 12214.493} C_VEL
LIN {X 0,Y 286.866,Z 1197.645,A -85,B 0,C 180,E1 12213.267,E2 12213.267} C_VEL
LIN {X 0,Y 299.288,Z 1188.104,A -85,B 0,C 180,E1 12210.586,E2 12210.586} C_VEL
LIN {X 0,Y 311.212,Z 1177.775,A -85,B 0,C 180,E1 12208.419,E2 12208.419} C_VEL
LIN {X 0,Y 323.906,Z 1165.438,A -85,B 0,C 180,E1 12206.456,E2 12206.456} C_VEL
LIN {X 0,Y 324.54,Z 1164.783,A -85,B 0,C 180,E1 12206.325,E2 12206.325} C_VEL
LIN {X 0,Y 310.273,Z 1179.989,A -85,B 0,C 180,E1 12204.296,E2 12204.296} C_VEL
LIN {X 0,Y 295.256,Z 1194.682,A -85,B 0,C 180,E1 12201.703,E2 12201.703} C_VEL
LIN {X 0,Y 280.987,Z 1207.847,A -85,B 0,C 180,E1 12198.658,E2 12198.658} C_VEL
LIN {X 0,Y 265.53,Z 1221.401,A -85,B 0,C 180,E1 12194.455,E2 12194.455} C_VEL
LIN {X 0,Y 252.721,Z 1232.291,A -85,B 0,C 180,E1 12189.858,E2 12189.858} C_VEL
LIN {X 0,Y 242.556,Z 1240.996,A -85,B 0,C 180,E1 12184.955,E2 12184.955} C_VEL
LIN {X 0,Y 234.105,Z 1248.558,A -85,B 0,C 180,E1 12179.133,E2 12179.133} C_VEL
LIN {X 0,Y 228.497,Z 1254.095,A -85,B 0,C 180,E1 12172.917,E2 12172.917} C_VEL
LIN {X 0,Y 225.906,Z 1257.435,A -85,B 0,C 180,E1 12166.981,E2 12166.981} C_VEL
LIN {X 0,Y 225.579,Z 1258.474,A -85,B 0,C 180,E1 12164.5,E2 12164.5} C_VEL
LIN {X 0,Y 225.073,Z 1266.473,A -85,B 0,C 180,E1 12159.974,E2 12159.974} C_VEL
LIN {X 0,Y 225.125,Z 1272.98,A -85,B 0,C 180,E1 12155.348,E2 12155.348} C_VEL
LIN {X 0,Y 225.198,Z 1277.085,A -85,B 0,C 180,E1 12151.523,E2 12151.523} C_VEL
LIN {X 0,Y 224.971,Z 1279.913,A -85,B 0,C 180,E1 12147.959,E2 12147.959} C_VEL
LIN {X 0,Y 224.485,Z 1282.34,A -85,B 0,C 180,E1 12143.346,E2 12143.346} C_VEL
LIN {X 0,Y 224.673,Z 1283.599,A -85,B 0,C 180,E1 12137.662,E2 12137.662} C_VEL
LIN {X 0,Y 226.759,Z 1283.333,A -85,B 0,C 180,E1 12131.486,E2 12131.486} C_VEL
LIN {X 0,Y 231.5,Z 1281.213,A -85,B 0,C 180,E1 12125.228,E2 12125.228} C_VEL
LIN {X 0,Y 240.044,Z 1277.004,A -85,B 0,C 180,E1 12118.641,E2 12118.641} C_VEL
LIN {X 0,Y 252.027,Z 1271.022,A -85,B 0,C 180,E1 12112.623,E2 12112.623} C_VEL
LIN {X 0,Y 266.513,Z 1263.718,A -85,B 0,C 180,E1 12107.518,E2 12107.518} C_VEL
LIN {X 0,Y 283.201,Z 1255.277,A -85,B 0,C 180,E1 12103.163,E2 12103.163} C_VEL
LIN {X 0,Y 265.827,Z 1261.595,A -85,B 0,C 180,E1 12098.363,E2 12098.363} C_VEL
LIN {X 0,Y 251.168,Z 1266.234,A -85,B 0,C 180,E1 12092.78,E2 12092.78} C_VEL
LIN {X 0,Y 240.36,Z 1268.87,A -85,B 0,C 180,E1 12086.965,E2 12086.965} C_VEL
LIN {X 0,Y 232.687,Z 1269.739,A -85,B 0,C 180,E1 12080.896,E2 12080.896} C_VEL
LIN {X 0,Y 227.83,Z 1268.78,A -85,B 0,C 180,E1 12074.747,E2 12074.747} C_VEL
LIN {X 0,Y 225.307,Z 1266.186,A -85,B 0,C 180,E1 12068.678,E2 12068.678} C_VEL
LIN {X 0,Y 224.401,Z 1262.493,A -85,B 0,C 180,E1 12063.321,E2 12063.321} C_VEL
LIN {X 0,Y 224.204,Z 1257.678,A -85,B 0,C 180,E1 12058.467,E2 12058.467} C_VEL
LIN {X 0,Y 224.319,Z 1251.502,A -85,B 0,C 180,E1 12053.602,E2 12053.602} C_VEL
LIN {X 0,Y 224.876,Z 1244.033,A -85,B 0,C 180,E1 12048.977,E2 12048.977} C_VEL
LIN {X 0,Y 226.207,Z 1234.41,A -85,B 0,C 180,E1 12044.094,E2 12044.094} C_VEL
LIN {X 0,Y 228.365,Z 1223.484,A -85,B 0,C 180,E1 12039.496,E2 12039.496} C_VEL
LIN {X 0,Y 231.52,Z 1210.385,A -85,B 0,C 180,E1 12034.96,E2 12034.96} C_VEL
LIN {X 0,Y 235.455,Z 1195.854,A -85,B 0,C 180,E1 12030.767,E2 12030.767} C_VEL
LIN {X 0,Y 240.212,Z 1179.326,A -85,B 0,C 180,E1 12026.795,E2 12026.795} C_VEL
LIN {X 0,Y 245.451,Z 1161.349,A -85,B 0,C 180,E1 12023.213,E2 12023.213} C_VEL
LIN {X 0,Y 250.875,Z 1142.399,A -85,B 0,C 180,E1 12020.082,E2 12020.082} C_VEL
LIN {X 0,Y 256.452,Z 1121.884,A -85,B 0,C 180,E1 12017.28,E2 12017.28} C_VEL
